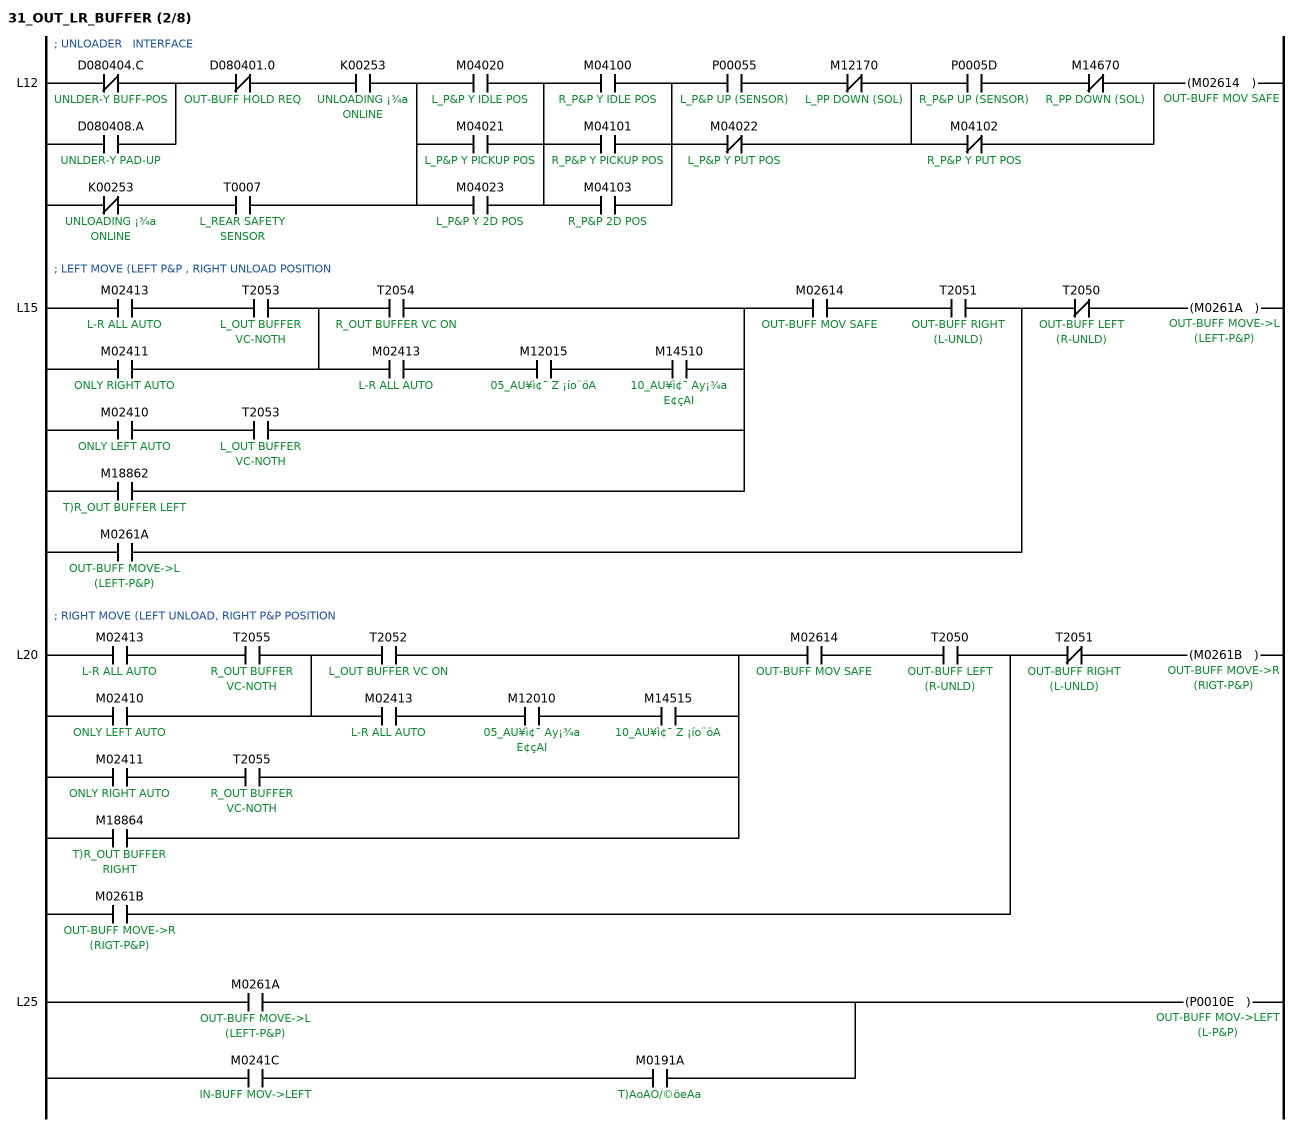
[picture p216: 31_OUT_LR_BUFFER rungs L12-L25]
//  UNLOADER   INTERFACE
; L12
LOAD NOT  D080404.C	// UNLDER-Y BUFF-POS
OR        D080408.A	// UNLDER-Y PAD-UP
AND NOT   D080401.0	// OUT-BUFF HOLD REQ
AND       K00253	// UNLOADING ¡¾a ONLINE
LOAD NOT  K00253	// UNLOADING ¡¾a ONLINE
AND       T0007	// L_REAR SAFETY SENSOR
OR LOAD
LOAD      M04020	// L_P&P Y IDLE POS
OR        M04021	// L_P&P Y PICKUP POS
OR        M04023	// L_P&P Y 2D POS
AND LOAD
LOAD      M04100	// R_P&P Y IDLE POS
OR        M04101	// R_P&P Y PICKUP POS
OR        M04103	// R_P&P 2D POS
AND LOAD
LOAD      P00055	// L_P&P UP (SENSOR)
AND NOT   M12170	// L_PP DOWN (SOL)
OR NOT    M04022	// L_P&P Y PUT POS
AND LOAD
LOAD      P0005D	// R_P&P UP (SENSOR)
AND NOT   M14670	// R_PP DOWN (SOL)
OR NOT    M04102	// R_P&P Y PUT POS
AND LOAD
OUT       M02614	// OUT-BUFF MOV SAFE
; L15
LOAD      M02413	// L-R ALL AUTO
AND       T2053	// L_OUT BUFFER VC-NOTH
OR        M02411	// ONLY RIGHT AUTO
LOAD      T2054	// R_OUT BUFFER VC ON
LOAD      M02413	// L-R ALL AUTO
AND       M12015	// 05_AU¥ì¢¯ Z ¡ío¨öA
AND       M14510	// 10_AU¥ì¢¯ Ay¡¾a E¢çAI
OR LOAD
AND LOAD
LOAD      M02410	// ONLY LEFT AUTO
AND       T2053	// L_OUT BUFFER VC-NOTH
OR LOAD
OR        M18862	// T)R_OUT BUFFER LEFT
AND       M02614	// OUT-BUFF MOV SAFE
AND       T2051	// OUT-BUFF RIGHT (L-UNLD)
OR        M0261A	// OUT-BUFF MOVE->L (LEFT-P&P)
AND NOT   T2050	// OUT-BUFF LEFT (R-UNLD)
OUT       M0261A	// OUT-BUFF MOVE->L (LEFT-P&P)
// output comment: LEFT MOVE (LEFT P&P , RIGHT UNLOAD POSITION
; L20
LOAD      M02413	// L-R ALL AUTO
AND       T2055	// R_OUT BUFFER VC-NOTH
OR        M02410	// ONLY LEFT AUTO
LOAD      T2052	// L_OUT BUFFER VC ON
LOAD      M02413	// L-R ALL AUTO
AND       M12010	// 05_AU¥ì¢¯ Ay¡¾a E¢çAI
AND       M14515	// 10_AU¥ì¢¯ Z ¡ío¨öA
OR LOAD
AND LOAD
LOAD      M02411	// ONLY RIGHT AUTO
AND       T2055	// R_OUT BUFFER VC-NOTH
OR LOAD
OR        M18864	// T)R_OUT BUFFER RIGHT
AND       M02614	// OUT-BUFF MOV SAFE
AND       T2050	// OUT-BUFF LEFT (R-UNLD)
OR        M0261B	// OUT-BUFF MOVE->R (RIGT-P&P)
AND NOT   T2051	// OUT-BUFF RIGHT (L-UNLD)
OUT       M0261B	// OUT-BUFF MOVE->R (RIGT-P&P)
// output comment: RIGHT MOVE (LEFT UNLOAD, RIGHT P&P POSITION
; L25
LOAD      M0261A	// OUT-BUFF MOVE->L (LEFT-P&P)
LOAD      M0241C	// IN-BUFF MOV->LEFT
AND       M0191A	// T)AoAO/©öeAa
OR LOAD
OUT       P0010E	// OUT-BUFF MOV->LEFT (L-P&P)

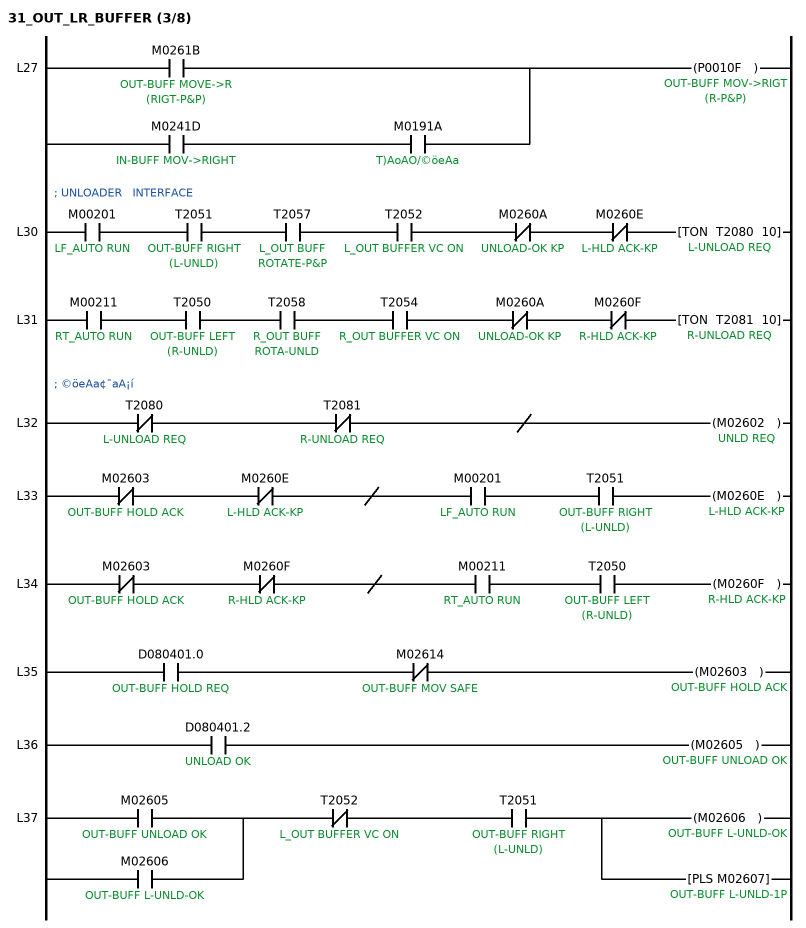
; L27
LOAD      M0261B	// OUT-BUFF MOVE->R (RIGT-P&P)
LOAD      M0241D	// IN-BUFF MOV->RIGHT
AND       M0191A	// T)AoAO/©öeAa
OR LOAD
OUT       P0010F	// OUT-BUFF MOV->RIGT (R-P&P)
//  UNLOADER   INTERFACE
; L30
LOAD      M00201	// LF_AUTO RUN
AND       T2051	// OUT-BUFF RIGHT (L-UNLD)
AND       T2057	// L_OUT BUFF ROTATE-P&P
AND       T2052	// L_OUT BUFFER VC ON
AND NOT   M0260A	// UNLOAD-OK KP
AND NOT   M0260E	// L-HLD ACK-KP
TON       T2080 10	// L-UNLOAD REQ
; L31
LOAD      M00211	// RT_AUTO RUN
AND       T2050	// OUT-BUFF LEFT (R-UNLD)
AND       T2058	// R_OUT BUFF ROTA-UNLD
AND       T2054	// R_OUT BUFFER VC ON
AND NOT   M0260A	// UNLOAD-OK KP
AND NOT   M0260F	// R-HLD ACK-KP
TON       T2081 10	// R-UNLOAD REQ
; L32
LOAD NOT  T2080	// L-UNLOAD REQ
AND NOT   T2081	// R-UNLOAD REQ
NOT
OUT       M02602	// UNLD REQ
// output comment: ©öeAa¢¯aA¡í
; L33
LOAD NOT  M02603	// OUT-BUFF HOLD ACK
AND NOT   M0260E	// L-HLD ACK-KP
NOT
AND       M00201	// LF_AUTO RUN
AND       T2051	// OUT-BUFF RIGHT (L-UNLD)
OUT       M0260E	// L-HLD ACK-KP
; L34
LOAD NOT  M02603	// OUT-BUFF HOLD ACK
AND NOT   M0260F	// R-HLD ACK-KP
NOT
AND       M00211	// RT_AUTO RUN
AND       T2050	// OUT-BUFF LEFT (R-UNLD)
OUT       M0260F	// R-HLD ACK-KP
; L35
LOAD      D080401.0	// OUT-BUFF HOLD REQ
AND NOT   M02614	// OUT-BUFF MOV SAFE
OUT       M02603	// OUT-BUFF HOLD ACK
; L36
LOAD      D080401.2	// UNLOAD OK
OUT       M02605	// OUT-BUFF UNLOAD OK
; L37
LOAD      M02605	// OUT-BUFF UNLOAD OK
OR        M02606	// OUT-BUFF L-UNLD-OK
AND NOT   T2052	// L_OUT BUFFER VC ON
AND       T2051	// OUT-BUFF RIGHT (L-UNLD)
OUT       M02606	// OUT-BUFF L-UNLD-OK
OUTP      M02607	// OUT-BUFF L-UNLD-1P

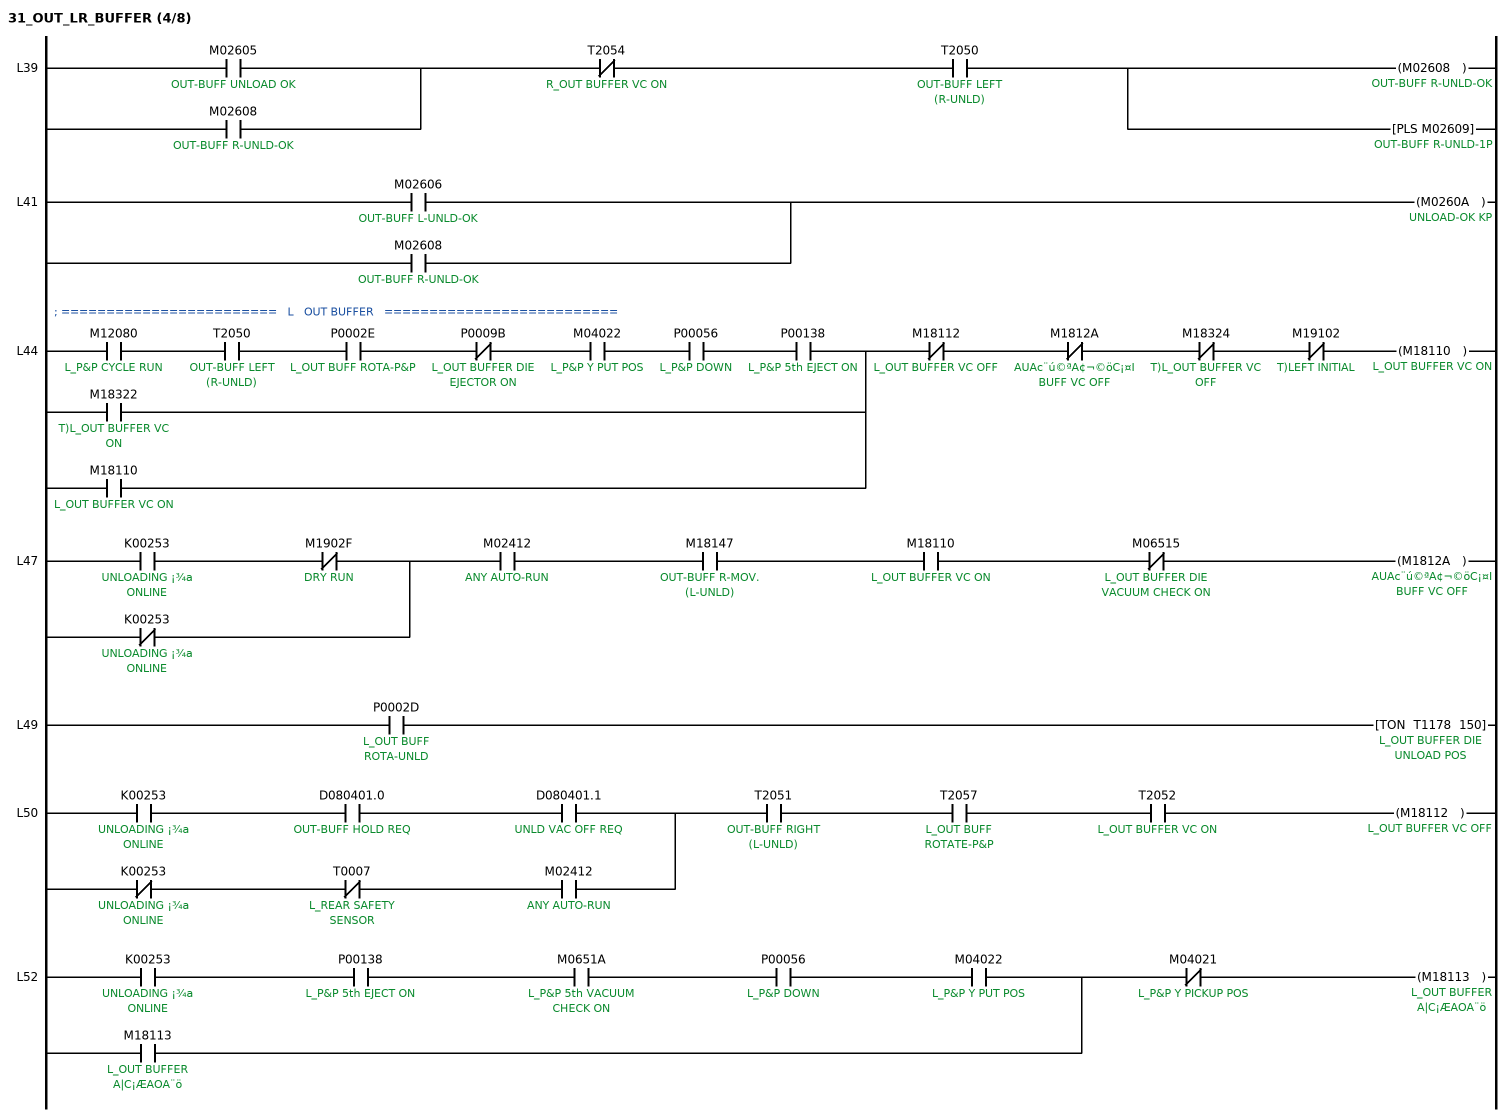
; L39
LOAD      M02605	// OUT-BUFF UNLOAD OK
OR        M02608	// OUT-BUFF R-UNLD-OK
AND NOT   T2054	// R_OUT BUFFER VC ON
AND       T2050	// OUT-BUFF LEFT (R-UNLD)
OUT       M02608	// OUT-BUFF R-UNLD-OK
OUTP      M02609	// OUT-BUFF R-UNLD-1P
; L41
LOAD      M02606	// OUT-BUFF L-UNLD-OK
OR        M02608	// OUT-BUFF R-UNLD-OK
OUT       M0260A	// UNLOAD-OK KP
// ========================   L   OUT BUFFER   ==========================
; L44
LOAD      M12080	// L_P&P CYCLE RUN
AND       T2050	// OUT-BUFF LEFT (R-UNLD)
AND       P0002E	// L_OUT BUFF ROTA-P&P
AND NOT   P0009B	// L_OUT BUFFER DIE EJECTOR ON
AND       M04022	// L_P&P Y PUT POS
AND       P00056	// L_P&P DOWN
AND       P00138	// L_P&P 5th EJECT ON
OR        M18322	// T)L_OUT BUFFER VC ON
OR        M18110	// L_OUT BUFFER VC ON
AND NOT   M18112	// L_OUT BUFFER VC OFF
AND NOT   M1812A	// AUAc¨ú©ªA¢¬©öC¡¤I BUFF VC OFF
AND NOT   M18324	// T)L_OUT BUFFER VC OFF
AND NOT   M19102	// T)LEFT INITIAL
OUT       M18110	// L_OUT BUFFER VC ON
; L47
LOAD      K00253	// UNLOADING ¡¾a ONLINE
AND NOT   M1902F	// DRY RUN
OR NOT    K00253	// UNLOADING ¡¾a ONLINE
AND       M02412	// ANY AUTO-RUN
AND       M18147	// OUT-BUFF R-MOV.  (L-UNLD)
AND       M18110	// L_OUT BUFFER VC ON
AND NOT   M06515	// L_OUT BUFFER DIE VACUUM CHECK ON
OUT       M1812A	// AUAc¨ú©ªA¢¬©öC¡¤I BUFF VC OFF
; L49
LOAD      P0002D	// L_OUT BUFF ROTA-UNLD
TON       T1178 150	// L_OUT BUFFER DIE UNLOAD POS
; L50
LOAD      K00253	// UNLOADING ¡¾a ONLINE
AND       D080401.0	// OUT-BUFF HOLD REQ
AND       D080401.1	// UNLD VAC OFF REQ
LOAD NOT  K00253	// UNLOADING ¡¾a ONLINE
AND NOT   T0007	// L_REAR SAFETY SENSOR
AND       M02412	// ANY AUTO-RUN
OR LOAD
AND       T2051	// OUT-BUFF RIGHT (L-UNLD)
AND       T2057	// L_OUT BUFF ROTATE-P&P
AND       T2052	// L_OUT BUFFER VC ON
OUT       M18112	// L_OUT BUFFER VC OFF
; L52
LOAD      K00253	// UNLOADING ¡¾a ONLINE
AND       P00138	// L_P&P 5th EJECT ON
AND       M0651A	// L_P&P 5th VACUUM CHECK ON
AND       P00056	// L_P&P DOWN
AND       M04022	// L_P&P Y PUT POS
OR        M18113	// L_OUT BUFFER A|C¡ÆAOA¨ö
AND NOT   M04021	// L_P&P Y PICKUP POS
OUT       M18113	// L_OUT BUFFER A|C¡ÆAOA¨ö

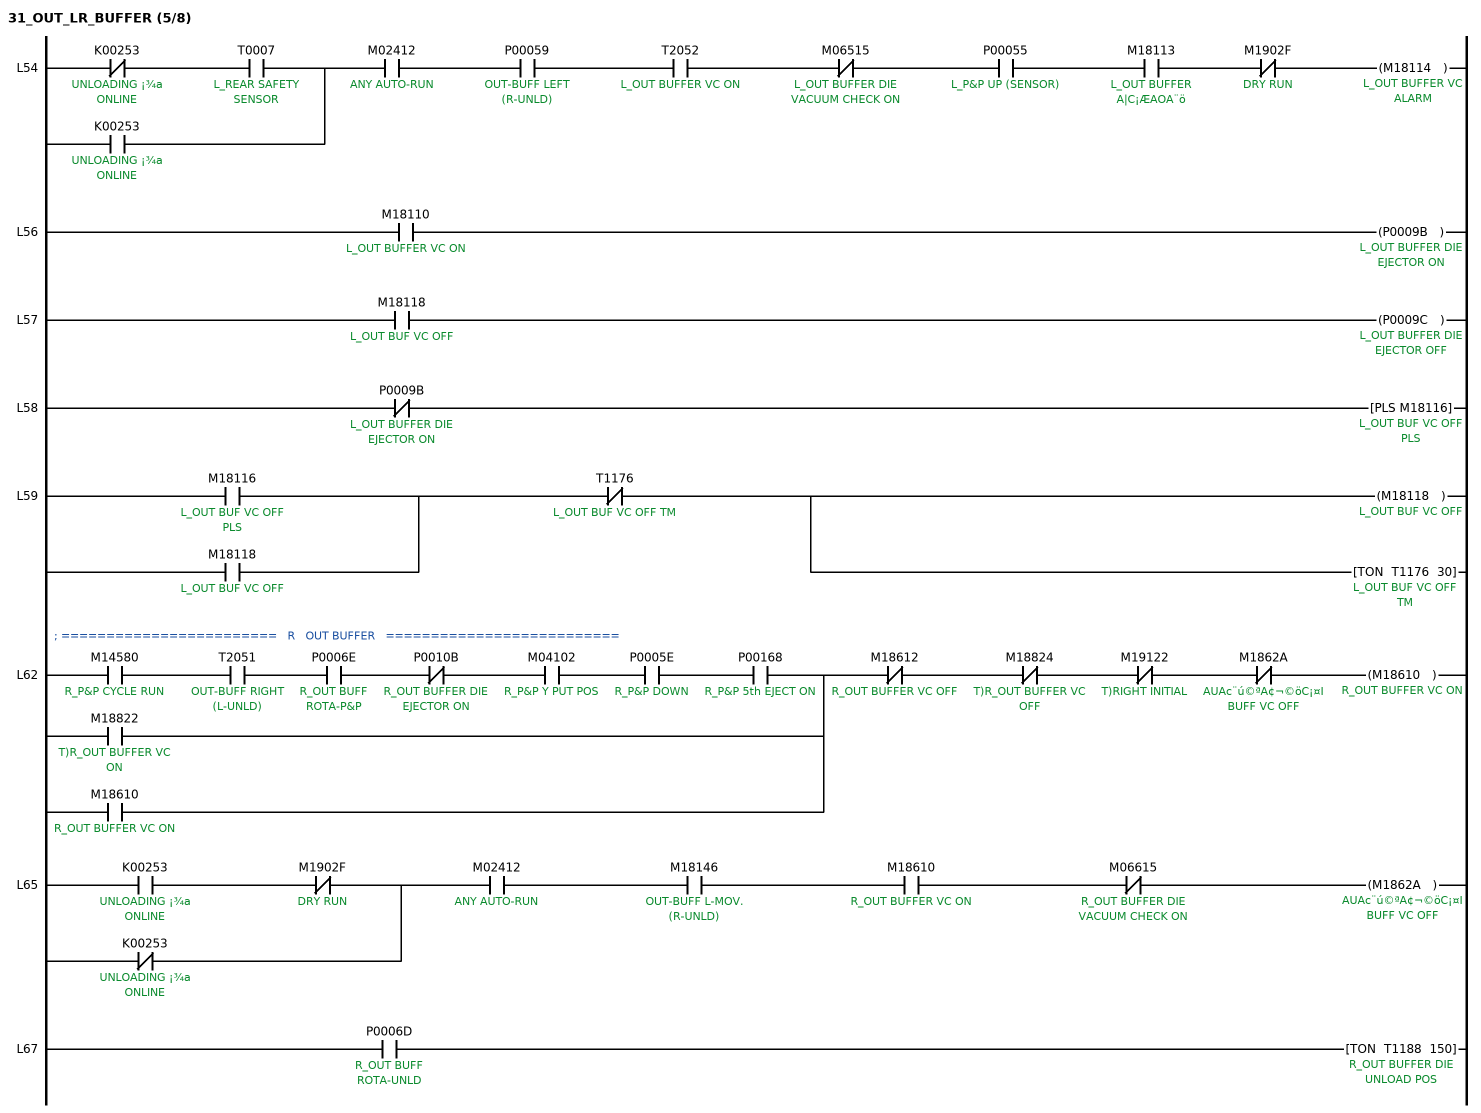
; L54
LOAD NOT  K00253	// UNLOADING ¡¾a ONLINE
AND       T0007	// L_REAR SAFETY SENSOR
OR        K00253	// UNLOADING ¡¾a ONLINE
AND       M02412	// ANY AUTO-RUN
AND       P00059	// OUT-BUFF LEFT (R-UNLD)
AND       T2052	// L_OUT BUFFER VC ON
AND NOT   M06515	// L_OUT BUFFER DIE VACUUM CHECK ON
AND       P00055	// L_P&P UP (SENSOR)
AND       M18113	// L_OUT BUFFER A|C¡ÆAOA¨ö
AND NOT   M1902F	// DRY RUN
OUT       M18114	// L_OUT BUFFER VC ALARM
; L56
LOAD      M18110	// L_OUT BUFFER VC ON
OUT       P0009B	// L_OUT BUFFER DIE EJECTOR ON
; L57
LOAD      M18118	// L_OUT BUF VC OFF
OUT       P0009C	// L_OUT BUFFER DIE EJECTOR OFF
; L58
LOAD NOT  P0009B	// L_OUT BUFFER DIE EJECTOR ON
OUTP      M18116	// L_OUT BUF VC OFF PLS
; L59
LOAD      M18116	// L_OUT BUF VC OFF PLS
OR        M18118	// L_OUT BUF VC OFF
AND NOT   T1176	// L_OUT BUF VC OFF TM
OUT       M18118	// L_OUT BUF VC OFF
TON       T1176 30	// L_OUT BUF VC OFF TM
// ========================   R   OUT BUFFER   ==========================
; L62
LOAD      M14580	// R_P&P CYCLE RUN
AND       T2051	// OUT-BUFF RIGHT (L-UNLD)
AND       P0006E	// R_OUT BUFF ROTA-P&P
AND NOT   P0010B	// R_OUT BUFFER DIE EJECTOR ON
AND       M04102	// R_P&P Y PUT POS
AND       P0005E	// R_P&P DOWN
AND       P00168	// R_P&P 5th EJECT ON
OR        M18822	// T)R_OUT BUFFER VC ON
OR        M18610	// R_OUT BUFFER VC ON
AND NOT   M18612	// R_OUT BUFFER VC OFF
AND NOT   M18824	// T)R_OUT BUFFER VC OFF
AND NOT   M19122	// T)RIGHT INITIAL
AND NOT   M1862A	// AUAc¨ú©ªA¢¬©öC¡¤I BUFF VC OFF
OUT       M18610	// R_OUT BUFFER VC ON
; L65
LOAD      K00253	// UNLOADING ¡¾a ONLINE
AND NOT   M1902F	// DRY RUN
OR NOT    K00253	// UNLOADING ¡¾a ONLINE
AND       M02412	// ANY AUTO-RUN
AND       M18146	// OUT-BUFF L-MOV.  (R-UNLD)
AND       M18610	// R_OUT BUFFER VC ON
AND NOT   M06615	// R_OUT BUFFER DIE VACUUM CHECK ON
OUT       M1862A	// AUAc¨ú©ªA¢¬©öC¡¤I BUFF VC OFF
; L67
LOAD      P0006D	// R_OUT BUFF ROTA-UNLD
TON       T1188 150	// R_OUT BUFFER DIE UNLOAD POS

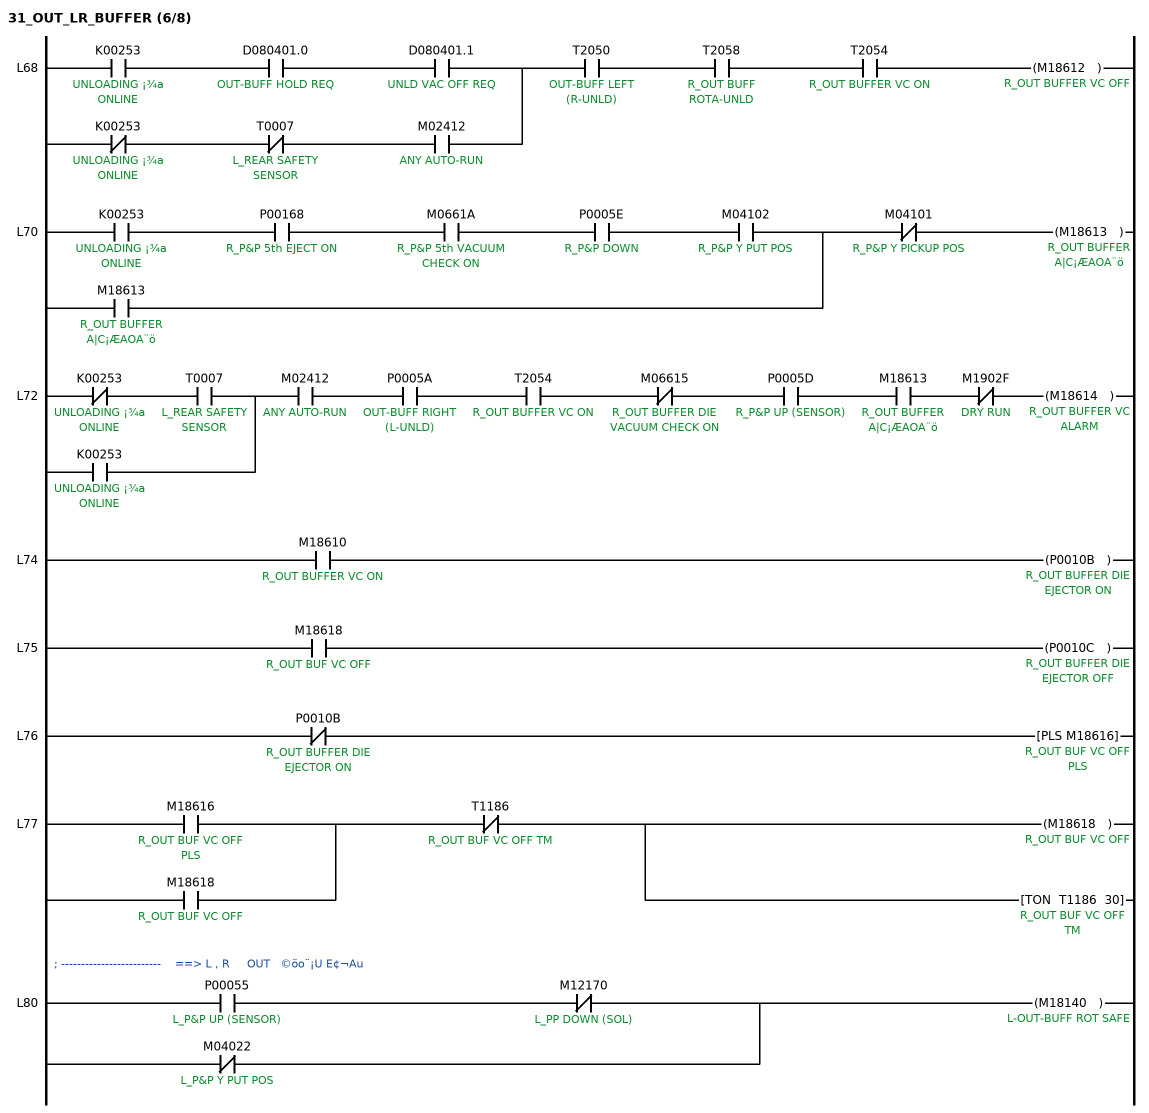
; L68
LOAD      K00253	// UNLOADING ¡¾a ONLINE
AND       D080401.0	// OUT-BUFF HOLD REQ
AND       D080401.1	// UNLD VAC OFF REQ
LOAD NOT  K00253	// UNLOADING ¡¾a ONLINE
AND NOT   T0007	// L_REAR SAFETY SENSOR
AND       M02412	// ANY AUTO-RUN
OR LOAD
AND       T2050	// OUT-BUFF LEFT (R-UNLD)
AND       T2058	// R_OUT BUFF ROTA-UNLD
AND       T2054	// R_OUT BUFFER VC ON
OUT       M18612	// R_OUT BUFFER VC OFF
; L70
LOAD      K00253	// UNLOADING ¡¾a ONLINE
AND       P00168	// R_P&P 5th EJECT ON
AND       M0661A	// R_P&P 5th VACUUM CHECK ON
AND       P0005E	// R_P&P DOWN
AND       M04102	// R_P&P Y PUT POS
OR        M18613	// R_OUT BUFFER A|C¡ÆAOA¨ö
AND NOT   M04101	// R_P&P Y PICKUP POS
OUT       M18613	// R_OUT BUFFER A|C¡ÆAOA¨ö
; L72
LOAD NOT  K00253	// UNLOADING ¡¾a ONLINE
AND       T0007	// L_REAR SAFETY SENSOR
OR        K00253	// UNLOADING ¡¾a ONLINE
AND       M02412	// ANY AUTO-RUN
AND       P0005A	// OUT-BUFF RIGHT (L-UNLD)
AND       T2054	// R_OUT BUFFER VC ON
AND NOT   M06615	// R_OUT BUFFER DIE VACUUM CHECK ON
AND       P0005D	// R_P&P UP (SENSOR)
AND       M18613	// R_OUT BUFFER A|C¡ÆAOA¨ö
AND NOT   M1902F	// DRY RUN
OUT       M18614	// R_OUT BUFFER VC ALARM
; L74
LOAD      M18610	// R_OUT BUFFER VC ON
OUT       P0010B	// R_OUT BUFFER DIE EJECTOR ON
; L75
LOAD      M18618	// R_OUT BUF VC OFF
OUT       P0010C	// R_OUT BUFFER DIE EJECTOR OFF
; L76
LOAD NOT  P0010B	// R_OUT BUFFER DIE EJECTOR ON
OUTP      M18616	// R_OUT BUF VC OFF PLS
; L77
LOAD      M18616	// R_OUT BUF VC OFF PLS
OR        M18618	// R_OUT BUF VC OFF
AND NOT   T1186	// R_OUT BUF VC OFF TM
OUT       M18618	// R_OUT BUF VC OFF
TON       T1186 30	// R_OUT BUF VC OFF TM
// -------------------------    ==> L , R     OUT   ©öo¨¡U E¢¬Au
; L80
LOAD      P00055	// L_P&P UP (SENSOR)
AND NOT   M12170	// L_PP DOWN (SOL)
OR NOT    M04022	// L_P&P Y PUT POS
OUT       M18140	// L-OUT-BUFF ROT SAFE

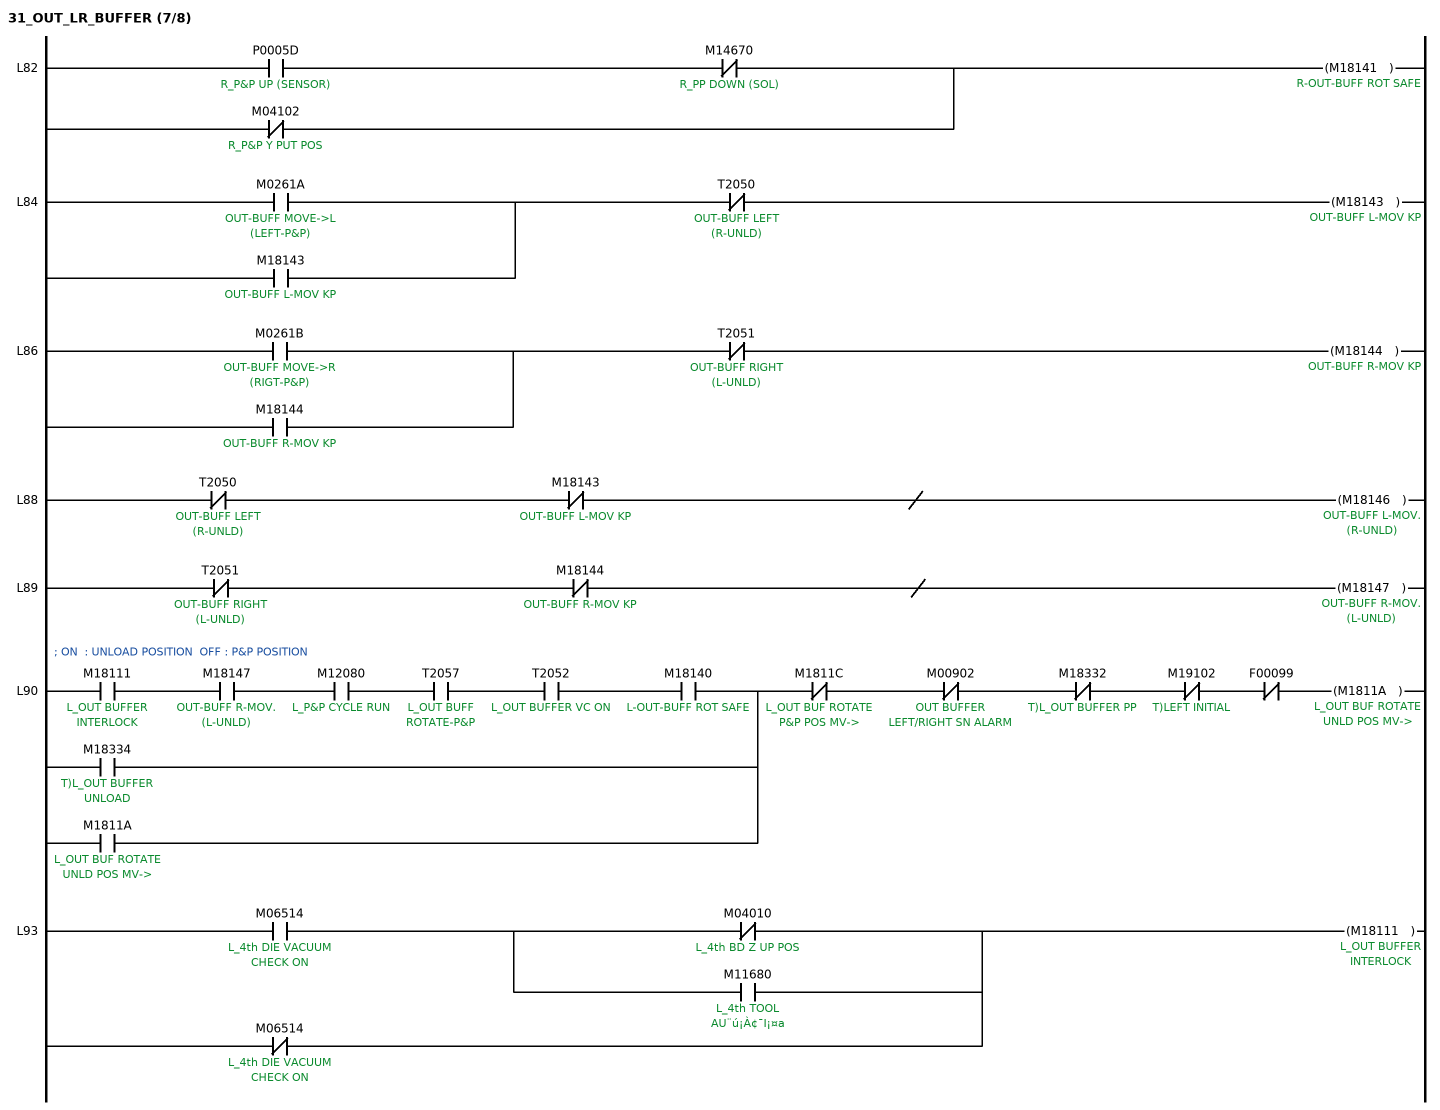
; L82
LOAD      P0005D	// R_P&P UP (SENSOR)
AND NOT   M14670	// R_PP DOWN (SOL)
OR NOT    M04102	// R_P&P Y PUT POS
OUT       M18141	// R-OUT-BUFF ROT SAFE
; L84
LOAD      M0261A	// OUT-BUFF MOVE->L (LEFT-P&P)
OR        M18143	// OUT-BUFF L-MOV KP
AND NOT   T2050	// OUT-BUFF LEFT (R-UNLD)
OUT       M18143	// OUT-BUFF L-MOV KP
; L86
LOAD      M0261B	// OUT-BUFF MOVE->R (RIGT-P&P)
OR        M18144	// OUT-BUFF R-MOV KP
AND NOT   T2051	// OUT-BUFF RIGHT (L-UNLD)
OUT       M18144	// OUT-BUFF R-MOV KP
; L88
LOAD NOT  T2050	// OUT-BUFF LEFT (R-UNLD)
AND NOT   M18143	// OUT-BUFF L-MOV KP
NOT
OUT       M18146	// OUT-BUFF L-MOV.  (R-UNLD)
; L89
LOAD NOT  T2051	// OUT-BUFF RIGHT (L-UNLD)
AND NOT   M18144	// OUT-BUFF R-MOV KP
NOT
OUT       M18147	// OUT-BUFF R-MOV.  (L-UNLD)
; L90
LOAD      M18111	// L_OUT BUFFER INTERLOCK
AND       M18147	// OUT-BUFF R-MOV.  (L-UNLD)
AND       M12080	// L_P&P CYCLE RUN
AND       T2057	// L_OUT BUFF ROTATE-P&P
AND       T2052	// L_OUT BUFFER VC ON
AND       M18140	// L-OUT-BUFF ROT SAFE
OR        M18334	// T)L_OUT BUFFER UNLOAD
OR        M1811A	// L_OUT BUF ROTATE UNLD POS MV->
AND NOT   M1811C	// L_OUT BUF ROTATE P&P POS MV->
AND NOT   M00902	// OUT BUFFER LEFT/RIGHT SN ALARM
AND NOT   M18332	// T)L_OUT BUFFER PP
AND NOT   M19102	// T)LEFT INITIAL
AND NOT   F00099
OUT       M1811A	// L_OUT BUF ROTATE UNLD POS MV->
// output comment: ON  : UNLOAD POSITION  OFF : P&P POSITION
; L93
LOAD      M06514	// L_4th DIE VACUUM CHECK ON
LOAD NOT  M04010	// L_4th BD Z UP POS
OR        M11680	// L_4th TOOL AU¨ú¡À¢¯I¡¤a
AND LOAD
OR NOT    M06514	// L_4th DIE VACUUM CHECK ON
OUT       M18111	// L_OUT BUFFER INTERLOCK

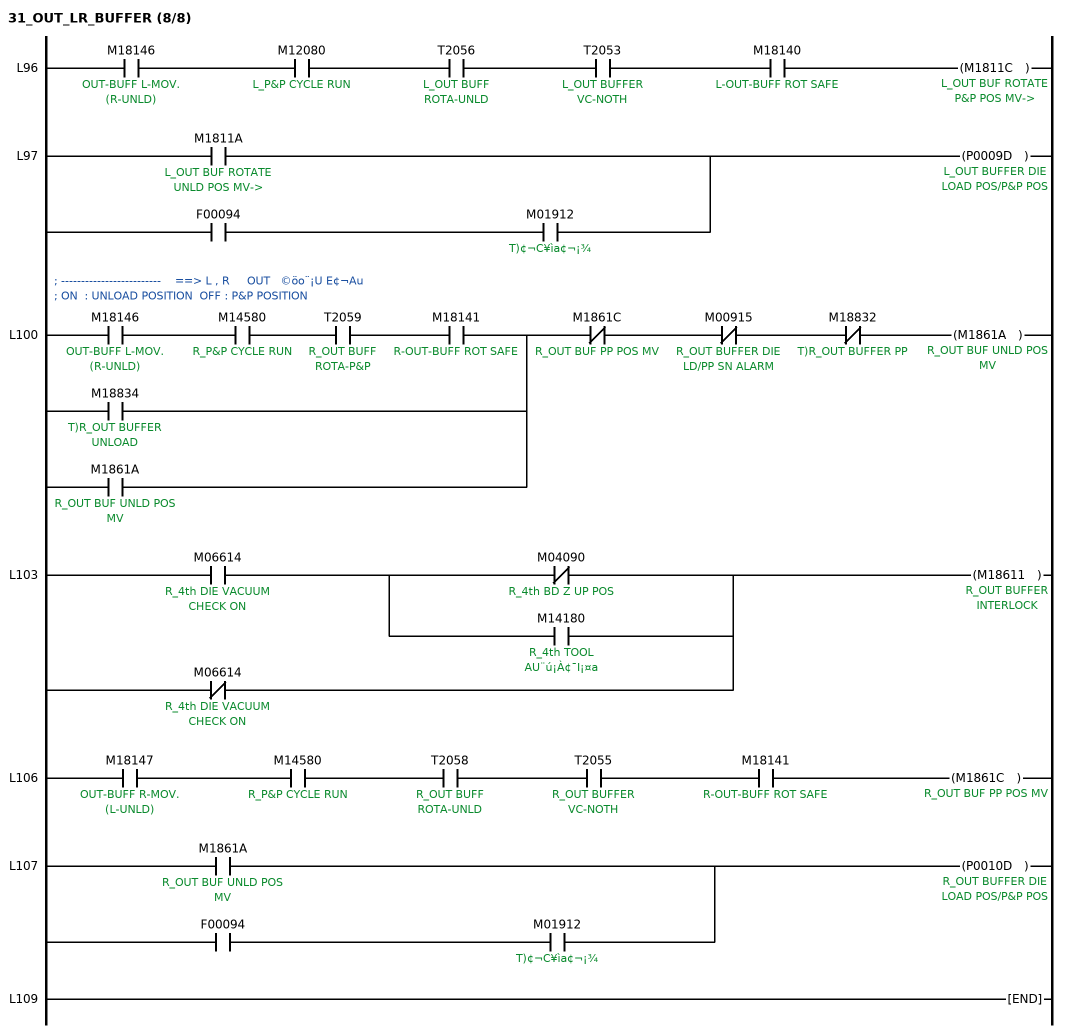
; L96
LOAD      M18146	// OUT-BUFF L-MOV.  (R-UNLD)
AND       M12080	// L_P&P CYCLE RUN
AND       T2056	// L_OUT BUFF ROTA-UNLD
AND       T2053	// L_OUT BUFFER VC-NOTH
AND       M18140	// L-OUT-BUFF ROT SAFE
OUT       M1811C	// L_OUT BUF ROTATE P&P POS MV->
; L97
LOAD      M1811A	// L_OUT BUF ROTATE UNLD POS MV->
LOAD      F00094
AND       M01912	// T)¢¬C¥ìa¢¬¡¾
OR LOAD
OUT       P0009D	// L_OUT BUFFER DIE LOAD POS/P&P POS
// -------------------------    ==> L , R     OUT   ©öo¨¡U E¢¬Au
; L100
LOAD      M18146	// OUT-BUFF L-MOV.  (R-UNLD)
AND       M14580	// R_P&P CYCLE RUN
AND       T2059	// R_OUT BUFF ROTA-P&P
AND       M18141	// R-OUT-BUFF ROT SAFE
OR        M18834	// T)R_OUT BUFFER UNLOAD
OR        M1861A	// R_OUT BUF UNLD POS MV
AND NOT   M1861C	// R_OUT BUF PP POS MV
AND NOT   M00915	// R_OUT BUFFER DIE LD/PP SN ALARM
AND NOT   M18832	// T)R_OUT BUFFER PP
OUT       M1861A	// R_OUT BUF UNLD POS MV
// output comment: ON  : UNLOAD POSITION  OFF : P&P POSITION
; L103
LOAD      M06614	// R_4th DIE VACUUM CHECK ON
LOAD NOT  M04090	// R_4th BD Z UP POS
OR        M14180	// R_4th TOOL AU¨ú¡À¢¯I¡¤a
AND LOAD
OR NOT    M06614	// R_4th DIE VACUUM CHECK ON
OUT       M18611	// R_OUT BUFFER INTERLOCK
; L106
LOAD      M18147	// OUT-BUFF R-MOV.  (L-UNLD)
AND       M14580	// R_P&P CYCLE RUN
AND       T2058	// R_OUT BUFF ROTA-UNLD
AND       T2055	// R_OUT BUFFER VC-NOTH
AND       M18141	// R-OUT-BUFF ROT SAFE
OUT       M1861C	// R_OUT BUF PP POS MV
; L107
LOAD      M1861A	// R_OUT BUF UNLD POS MV
LOAD      F00094
AND       M01912	// T)¢¬C¥ìa¢¬¡¾
OR LOAD
OUT       P0010D	// R_OUT BUFFER DIE LOAD POS/P&P POS
; L109
END

PROGRAM 40_2D_CODE (task: ¨ö¨¬A¥ì CA¡¤I¡¾¡¿¡¤¡Í)

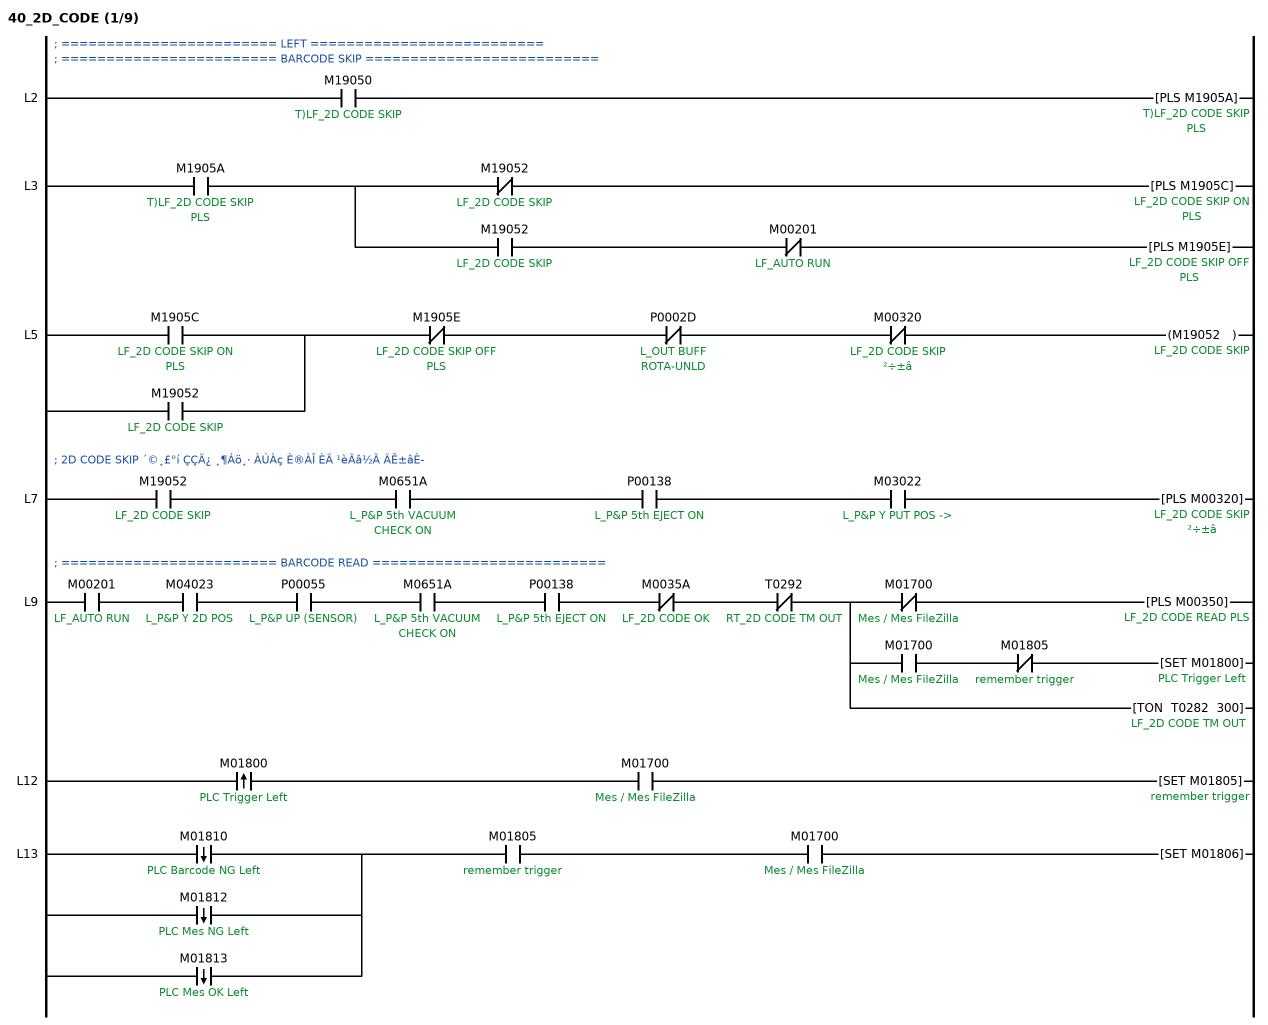
// ======================== LEFT ==========================
// ======================== BARCODE SKIP ==========================
; L2
LOAD      M19050	// T)LF_2D CODE SKIP
OUTP      M1905A	// T)LF_2D CODE SKIP PLS
; L3
LOAD      M1905A	// T)LF_2D CODE SKIP PLS
MPUSH
AND NOT   M19052	// LF_2D CODE SKIP
OUTP      M1905C	// LF_2D CODE SKIP ON PLS
MPOP
AND       M19052	// LF_2D CODE SKIP
AND NOT   M00201	// LF_AUTO RUN
OUTP      M1905E	// LF_2D CODE SKIP OFF PLS
; L5
LOAD      M1905C	// LF_2D CODE SKIP ON PLS
OR        M19052	// LF_2D CODE SKIP
AND NOT   M1905E	// LF_2D CODE SKIP OFF PLS
AND NOT   P0002D	// L_OUT BUFF ROTA-UNLD
AND NOT   M00320	// LF_2D CODE SKIP ²÷±â
OUT       M19052	// LF_2D CODE SKIP
; L7
LOAD      M19052	// LF_2D CODE SKIP
AND       M0651A	// L_P&P 5th VACUUM CHECK ON
AND       P00138	// L_P&P 5th EJECT ON
AND       M03022	// L_P&P Y PUT POS ->
OUTP      M00320	// LF_2D CODE SKIP ²÷±â
// output comment: 2D CODE SKIP ´©¸£°í ÇÇÄ¿ ¸¶Áö¸· ÀÚÀç È®ÀÎ ÈÄ ¹èÃâ½Ã ÃÊ±âÈ­
// ======================== BARCODE READ ==========================
; L9
LOAD      M00201	// LF_AUTO RUN
AND       M04023	// L_P&P Y 2D POS
AND       P00055	// L_P&P UP (SENSOR)
AND       M0651A	// L_P&P 5th VACUUM CHECK ON
AND       P00138	// L_P&P 5th EJECT ON
AND NOT   M0035A	// LF_2D CODE OK
AND NOT   T0292	// RT_2D CODE TM OUT
MPUSH
AND NOT   M01700	// Mes / Mes FileZilla
OUTP      M00350	// LF_2D CODE READ PLS
MLOAD
AND       M01700	// Mes / Mes FileZilla
AND NOT   M01805	// remember trigger
SET       M01800	// PLC Trigger Left
MPOP
TON       T0282 300	// LF_2D CODE TM OUT
; L12
LOADP     M01800	// PLC Trigger Left
AND       M01700	// Mes / Mes FileZilla
SET       M01805	// remember trigger
; L13
LOADN     M01810	// PLC Barcode NG Left
ORN       M01812	// PLC Mes NG Left
ORN       M01813	// PLC Mes OK Left
AND       M01805	// remember trigger
AND       M01700	// Mes / Mes FileZilla
SET       M01806

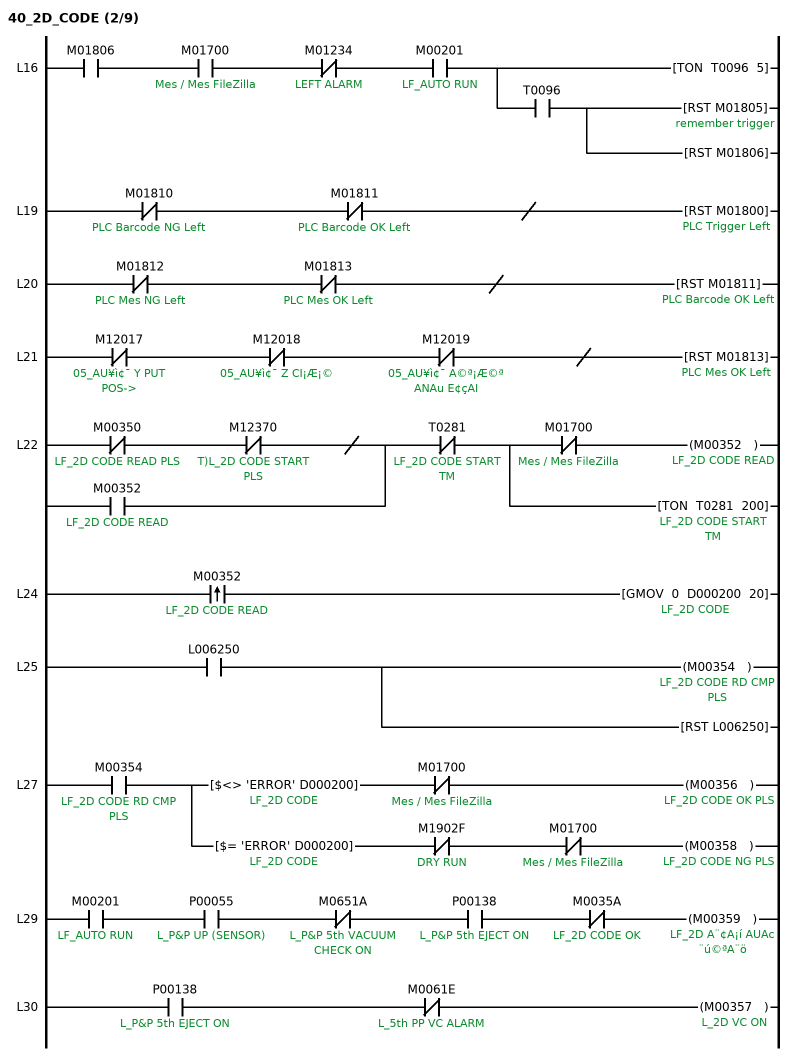
; L16
LOAD      M01806
AND       M01700	// Mes / Mes FileZilla
AND NOT   M01234	// LEFT ALARM
AND       M00201	// LF_AUTO RUN
TON       T0096 5
AND       T0096
RST       M01805	// remember trigger
RST       M01806
; L19
LOAD NOT  M01810	// PLC Barcode NG Left
AND NOT   M01811	// PLC Barcode OK Left
NOT
RST       M01800	// PLC Trigger Left
; L20
LOAD NOT  M01812	// PLC Mes NG Left
AND NOT   M01813	// PLC Mes OK Left
NOT
RST       M01811	// PLC Barcode OK Left
; L21
LOAD NOT  M12017	// 05_AU¥ì¢¯ Y PUT POS->
AND NOT   M12018	// 05_AU¥ì¢¯ Z CI¡Æ¡©
AND NOT   M12019	// 05_AU¥ì¢¯ A©ª¡Æ©ª ANAu E¢çAI
NOT
RST       M01813	// PLC Mes OK Left
; L22
LOAD NOT  M00350	// LF_2D CODE READ PLS
AND NOT   M12370	// T)L_2D CODE START PLS
NOT
OR        M00352	// LF_2D CODE READ
AND NOT   T0281	// LF_2D CODE START TM
MPUSH
AND NOT   M01700	// Mes / Mes FileZilla
OUT       M00352	// LF_2D CODE READ
MPOP
TON       T0281 200	// LF_2D CODE START TM
; L24
LOADP     M00352	// LF_2D CODE READ
GMOV      0 D000200 20	// LF_2D CODE
; L25
LOAD      L006250
OUT       M00354	// LF_2D CODE RD CMP PLS
RST       L006250
; L27
LOAD      M00354	// LF_2D CODE RD CMP PLS
MPUSH
AND$<>    'ERROR' D000200	// LF_2D CODE
AND NOT   M01700	// Mes / Mes FileZilla
OUT       M00356	// LF_2D CODE OK PLS
MPOP
AND$=     'ERROR' D000200	// LF_2D CODE
AND NOT   M1902F	// DRY RUN
AND NOT   M01700	// Mes / Mes FileZilla
OUT       M00358	// LF_2D CODE NG PLS
; L29
LOAD      M00201	// LF_AUTO RUN
AND       P00055	// L_P&P UP (SENSOR)
AND NOT   M0651A	// L_P&P 5th VACUUM CHECK ON
AND       P00138	// L_P&P 5th EJECT ON
AND NOT   M0035A	// LF_2D CODE OK
OUT       M00359	// LF_2D A¨¢A¡í AUAc ¨ú©ªA¨ö
; L30
LOAD      P00138	// L_P&P 5th EJECT ON
AND NOT   M0061E	// L_5th PP VC ALARM
OUT       M00357	// L_2D VC ON

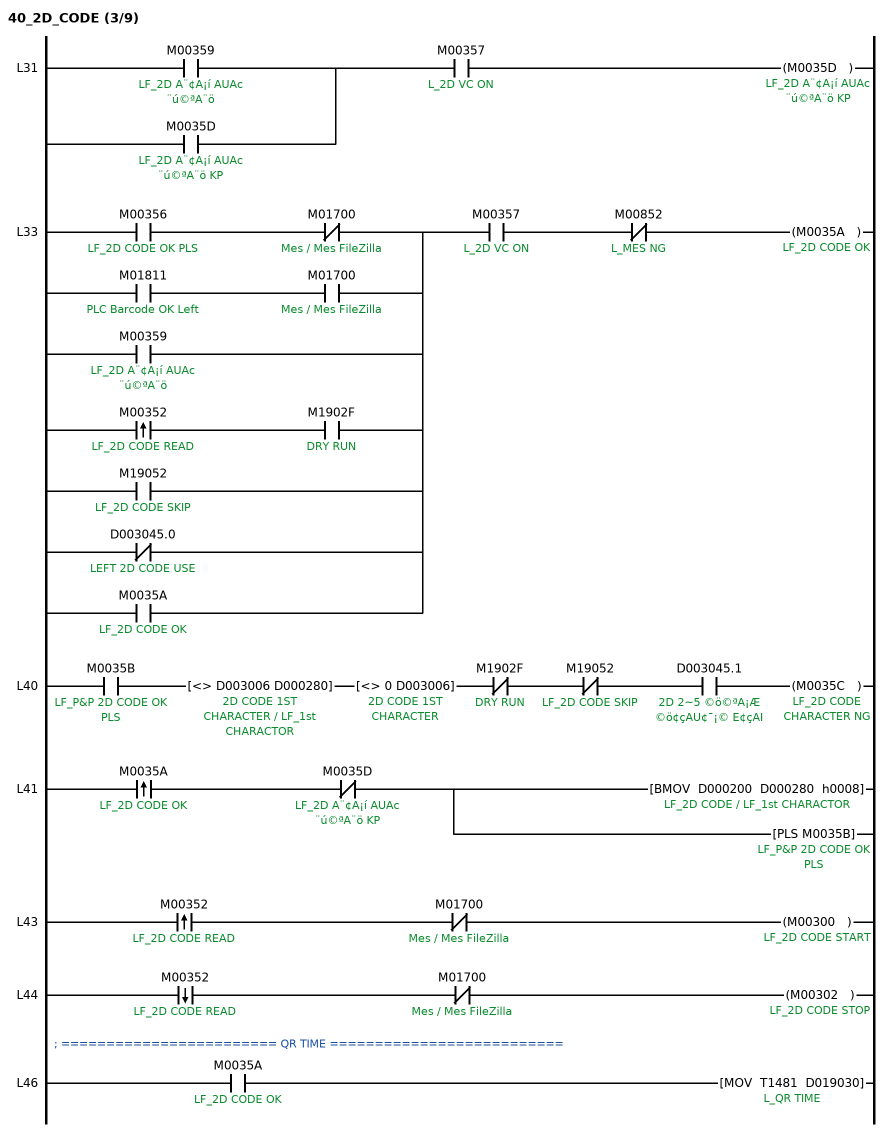
; L31
LOAD      M00359	// LF_2D A¨¢A¡í AUAc ¨ú©ªA¨ö
OR        M0035D	// LF_2D A¨¢A¡í AUAc ¨ú©ªA¨ö KP
AND       M00357	// L_2D VC ON
OUT       M0035D	// LF_2D A¨¢A¡í AUAc ¨ú©ªA¨ö KP
; L33
LOAD      M00356	// LF_2D CODE OK PLS
AND NOT   M01700	// Mes / Mes FileZilla
LOAD      M01811	// PLC Barcode OK Left
AND       M01700	// Mes / Mes FileZilla
OR LOAD
OR        M00359	// LF_2D A¨¢A¡í AUAc ¨ú©ªA¨ö
LOADP     M00352	// LF_2D CODE READ
AND       M1902F	// DRY RUN
OR LOAD
OR        M19052	// LF_2D CODE SKIP
OR NOT    D003045.0	// LEFT 2D CODE USE
OR        M0035A	// LF_2D CODE OK
AND       M00357	// L_2D VC ON
AND NOT   M00852	// L_MES NG
OUT       M0035A	// LF_2D CODE OK
; L40
LOAD      M0035B	// LF_P&P 2D CODE OK PLS
AND<>     D003006 D000280	// 2D CODE 1ST CHARACTER / LF_1st CHARACTOR
AND<>     0 D003006	// 2D CODE 1ST CHARACTER
AND NOT   M1902F	// DRY RUN
AND NOT   M19052	// LF_2D CODE SKIP
AND       D003045.1	// 2D 2~5 ©ö©ªA¡Æ ©ö¢çAU¢¯¡© E¢çAI
OUT       M0035C	// LF_2D CODE CHARACTER NG
; L41
LOADP     M0035A	// LF_2D CODE OK
AND NOT   M0035D	// LF_2D A¨¢A¡í AUAc ¨ú©ªA¨ö KP
BMOV      D000200 D000280 h0008	// LF_2D CODE / LF_1st CHARACTOR
OUTP      M0035B	// LF_P&P 2D CODE OK PLS
; L43
LOADP     M00352	// LF_2D CODE READ
AND NOT   M01700	// Mes / Mes FileZilla
OUT       M00300	// LF_2D CODE START
; L44
LOADN     M00352	// LF_2D CODE READ
AND NOT   M01700	// Mes / Mes FileZilla
OUT       M00302	// LF_2D CODE STOP
// ======================== QR TIME ==========================
; L46
LOAD      M0035A	// LF_2D CODE OK
MOV       T1481 D019030	// L_QR TIME

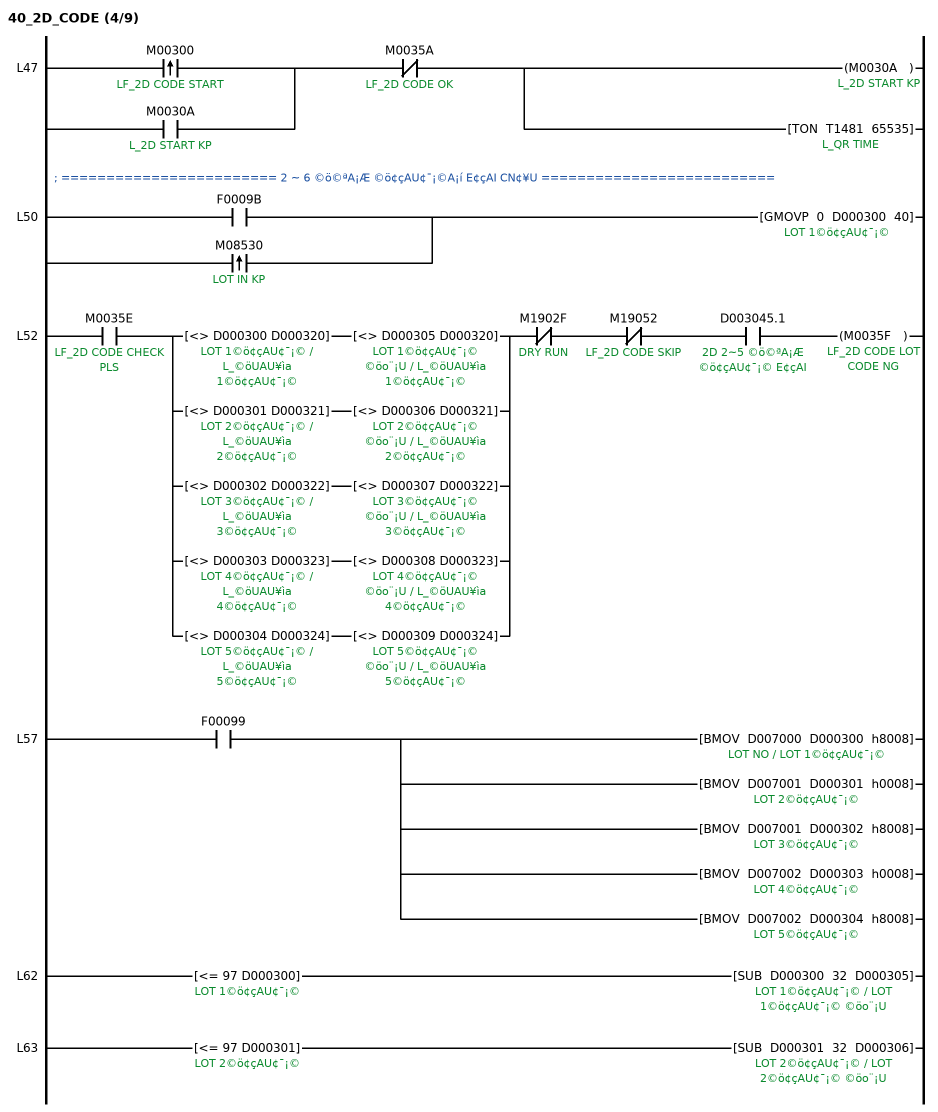
; L47
LOADP     M00300	// LF_2D CODE START
OR        M0030A	// L_2D START KP
AND NOT   M0035A	// LF_2D CODE OK
OUT       M0030A	// L_2D START KP
TON       T1481 65535	// L_QR TIME
// ======================== 2 ~ 6 ©ö©ªA¡Æ ©ö¢çAU¢¯¡©A¡í E¢çAI CN¢¥U ==========================
; L50
LOAD      F0009B
ORP       M08530	// LOT IN KP
GMOVP     0 D000300 40	// LOT 1©ö¢çAU¢¯¡©
; L52
LOAD      M0035E	// LF_2D CODE CHECK PLS
LOAD<>    D000300 D000320	// LOT 1©ö¢çAU¢¯¡© / L_©öUAU¥ìa 1©ö¢çAU¢¯¡©
AND<>     D000305 D000320	// LOT 1©ö¢çAU¢¯¡© ©öo¨¡U / L_©öUAU¥ìa 1©ö¢çAU¢¯¡©
LOAD<>    D000301 D000321	// LOT 2©ö¢çAU¢¯¡© / L_©öUAU¥ìa 2©ö¢çAU¢¯¡©
AND<>     D000306 D000321	// LOT 2©ö¢çAU¢¯¡© ©öo¨¡U / L_©öUAU¥ìa 2©ö¢çAU¢¯¡©
OR LOAD
LOAD<>    D000302 D000322	// LOT 3©ö¢çAU¢¯¡© / L_©öUAU¥ìa 3©ö¢çAU¢¯¡©
AND<>     D000307 D000322	// LOT 3©ö¢çAU¢¯¡© ©öo¨¡U / L_©öUAU¥ìa 3©ö¢çAU¢¯¡©
OR LOAD
LOAD<>    D000303 D000323	// LOT 4©ö¢çAU¢¯¡© / L_©öUAU¥ìa 4©ö¢çAU¢¯¡©
AND<>     D000308 D000323	// LOT 4©ö¢çAU¢¯¡© ©öo¨¡U / L_©öUAU¥ìa 4©ö¢çAU¢¯¡©
OR LOAD
LOAD<>    D000304 D000324	// LOT 5©ö¢çAU¢¯¡© / L_©öUAU¥ìa 5©ö¢çAU¢¯¡©
AND<>     D000309 D000324	// LOT 5©ö¢çAU¢¯¡© ©öo¨¡U / L_©öUAU¥ìa 5©ö¢çAU¢¯¡©
OR LOAD
AND LOAD
AND NOT   M1902F	// DRY RUN
AND NOT   M19052	// LF_2D CODE SKIP
AND       D003045.1	// 2D 2~5 ©ö©ªA¡Æ ©ö¢çAU¢¯¡© E¢çAI
OUT       M0035F	// LF_2D CODE LOT CODE NG
; L57
LOAD      F00099
BMOV      D007000 D000300 h8008	// LOT NO / LOT 1©ö¢çAU¢¯¡©
BMOV      D007001 D000301 h0008	// LOT 2©ö¢çAU¢¯¡©
BMOV      D007001 D000302 h8008	// LOT 3©ö¢çAU¢¯¡©
BMOV      D007002 D000303 h0008	// LOT 4©ö¢çAU¢¯¡©
BMOV      D007002 D000304 h8008	// LOT 5©ö¢çAU¢¯¡©
; L62
LOAD<=    97 D000300	// LOT 1©ö¢çAU¢¯¡©
SUB       D000300 32 D000305	// LOT 1©ö¢çAU¢¯¡© / LOT 1©ö¢çAU¢¯¡© ©öo¨¡U
; L63
LOAD<=    97 D000301	// LOT 2©ö¢çAU¢¯¡©
SUB       D000301 32 D000306	// LOT 2©ö¢çAU¢¯¡© / LOT 2©ö¢çAU¢¯¡© ©öo¨¡U

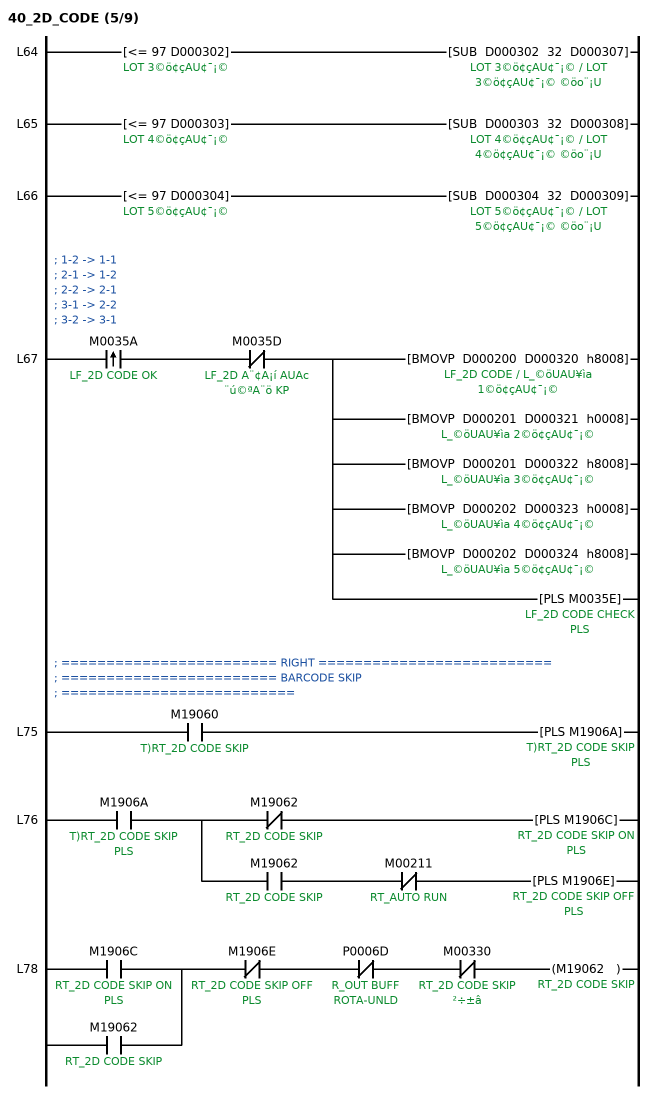
; L64
LOAD<=    97 D000302	// LOT 3©ö¢çAU¢¯¡©
SUB       D000302 32 D000307	// LOT 3©ö¢çAU¢¯¡© / LOT 3©ö¢çAU¢¯¡© ©öo¨¡U
; L65
LOAD<=    97 D000303	// LOT 4©ö¢çAU¢¯¡©
SUB       D000303 32 D000308	// LOT 4©ö¢çAU¢¯¡© / LOT 4©ö¢çAU¢¯¡© ©öo¨¡U
; L66
LOAD<=    97 D000304	// LOT 5©ö¢çAU¢¯¡©
SUB       D000304 32 D000309	// LOT 5©ö¢çAU¢¯¡© / LOT 5©ö¢çAU¢¯¡© ©öo¨¡U
; L67
LOADP     M0035A	// LF_2D CODE OK
AND NOT   M0035D	// LF_2D A¨¢A¡í AUAc ¨ú©ªA¨ö KP
BMOVP     D000200 D000320 h8008	// LF_2D CODE / L_©öUAU¥ìa 1©ö¢çAU¢¯¡©
BMOVP     D000201 D000321 h0008	// L_©öUAU¥ìa 2©ö¢çAU¢¯¡©
BMOVP     D000201 D000322 h8008	// L_©öUAU¥ìa 3©ö¢çAU¢¯¡©
BMOVP     D000202 D000323 h0008	// L_©öUAU¥ìa 4©ö¢çAU¢¯¡©
BMOVP     D000202 D000324 h8008	// L_©öUAU¥ìa 5©ö¢çAU¢¯¡©
OUTP      M0035E	// LF_2D CODE CHECK PLS
// output comment: 1-2 -> 1-1
// output comment: 2-1 -> 1-2
// output comment: 2-2 -> 2-1
// output comment: 3-1 -> 2-2
// output comment: 3-2 -> 3-1
// ======================== RIGHT ==========================
// ======================== BARCODE SKIP ==========================
; L75
LOAD      M19060	// T)RT_2D CODE SKIP
OUTP      M1906A	// T)RT_2D CODE SKIP PLS
; L76
LOAD      M1906A	// T)RT_2D CODE SKIP PLS
MPUSH
AND NOT   M19062	// RT_2D CODE SKIP
OUTP      M1906C	// RT_2D CODE SKIP ON PLS
MPOP
AND       M19062	// RT_2D CODE SKIP
AND NOT   M00211	// RT_AUTO RUN
OUTP      M1906E	// RT_2D CODE SKIP OFF PLS
; L78
LOAD      M1906C	// RT_2D CODE SKIP ON PLS
OR        M19062	// RT_2D CODE SKIP
AND NOT   M1906E	// RT_2D CODE SKIP OFF PLS
AND NOT   P0006D	// R_OUT BUFF ROTA-UNLD
AND NOT   M00330	// RT_2D CODE SKIP ²÷±â
OUT       M19062	// RT_2D CODE SKIP

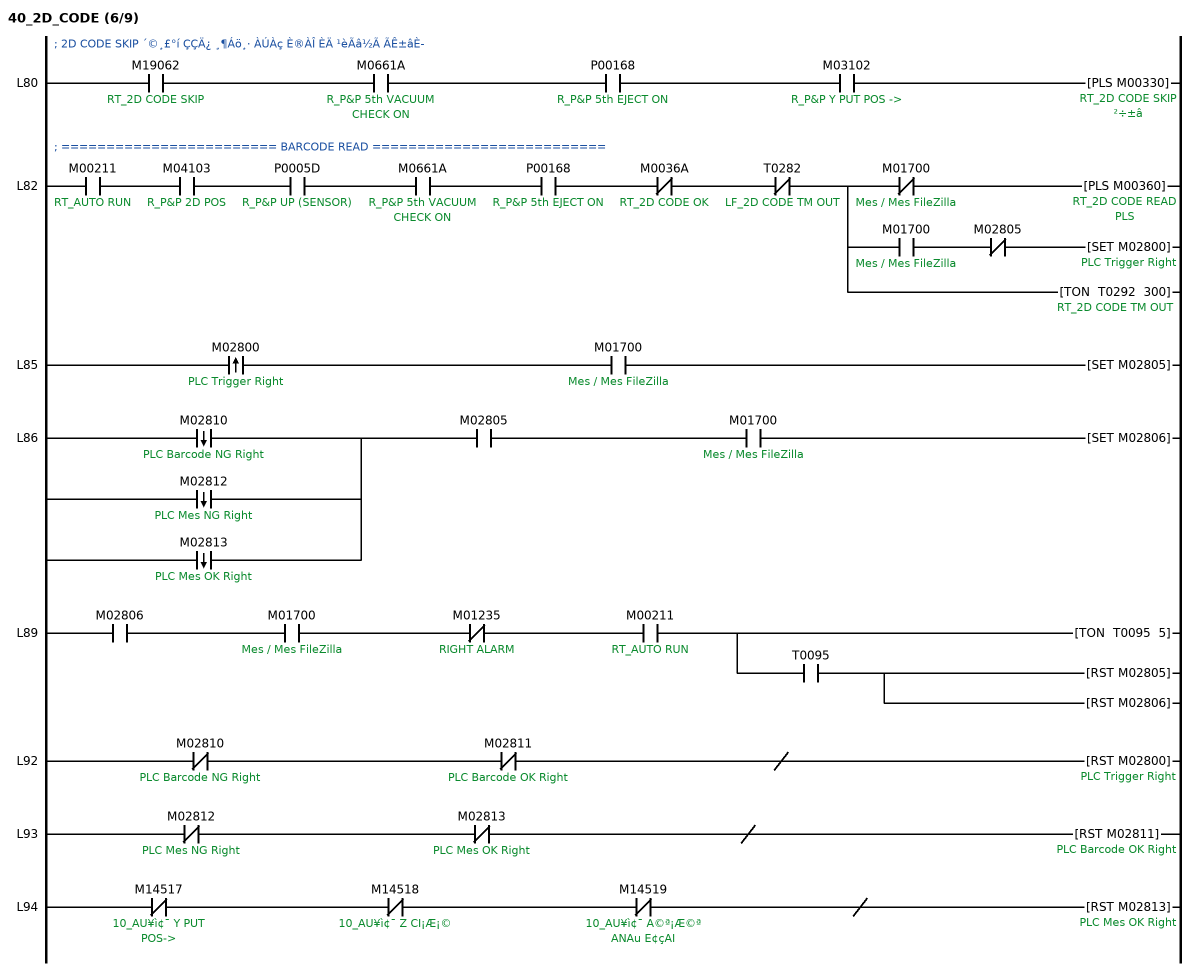
; L80
LOAD      M19062	// RT_2D CODE SKIP
AND       M0661A	// R_P&P 5th VACUUM CHECK ON
AND       P00168	// R_P&P 5th EJECT ON
AND       M03102	// R_P&P Y PUT POS ->
OUTP      M00330	// RT_2D CODE SKIP ²÷±â
// output comment: 2D CODE SKIP ´©¸£°í ÇÇÄ¿ ¸¶Áö¸· ÀÚÀç È®ÀÎ ÈÄ ¹èÃâ½Ã ÃÊ±âÈ­
// ======================== BARCODE READ ==========================
; L82
LOAD      M00211	// RT_AUTO RUN
AND       M04103	// R_P&P 2D POS
AND       P0005D	// R_P&P UP (SENSOR)
AND       M0661A	// R_P&P 5th VACUUM CHECK ON
AND       P00168	// R_P&P 5th EJECT ON
AND NOT   M0036A	// RT_2D CODE OK
AND NOT   T0282	// LF_2D CODE TM OUT
MPUSH
AND NOT   M01700	// Mes / Mes FileZilla
OUTP      M00360	// RT_2D CODE READ PLS
MLOAD
AND       M01700	// Mes / Mes FileZilla
AND NOT   M02805
SET       M02800	// PLC Trigger Right
MPOP
TON       T0292 300	// RT_2D CODE TM OUT
; L85
LOADP     M02800	// PLC Trigger Right
AND       M01700	// Mes / Mes FileZilla
SET       M02805
; L86
LOADN     M02810	// PLC Barcode NG Right
ORN       M02812	// PLC Mes NG Right
ORN       M02813	// PLC Mes OK Right
AND       M02805
AND       M01700	// Mes / Mes FileZilla
SET       M02806
; L89
LOAD      M02806
AND       M01700	// Mes / Mes FileZilla
AND NOT   M01235	// RIGHT ALARM
AND       M00211	// RT_AUTO RUN
TON       T0095 5
AND       T0095
RST       M02805
RST       M02806
; L92
LOAD NOT  M02810	// PLC Barcode NG Right
AND NOT   M02811	// PLC Barcode OK Right
NOT
RST       M02800	// PLC Trigger Right
; L93
LOAD NOT  M02812	// PLC Mes NG Right
AND NOT   M02813	// PLC Mes OK Right
NOT
RST       M02811	// PLC Barcode OK Right
; L94
LOAD NOT  M14517	// 10_AU¥ì¢¯ Y PUT POS->
AND NOT   M14518	// 10_AU¥ì¢¯ Z CI¡Æ¡©
AND NOT   M14519	// 10_AU¥ì¢¯ A©ª¡Æ©ª ANAu E¢çAI
NOT
RST       M02813	// PLC Mes OK Right

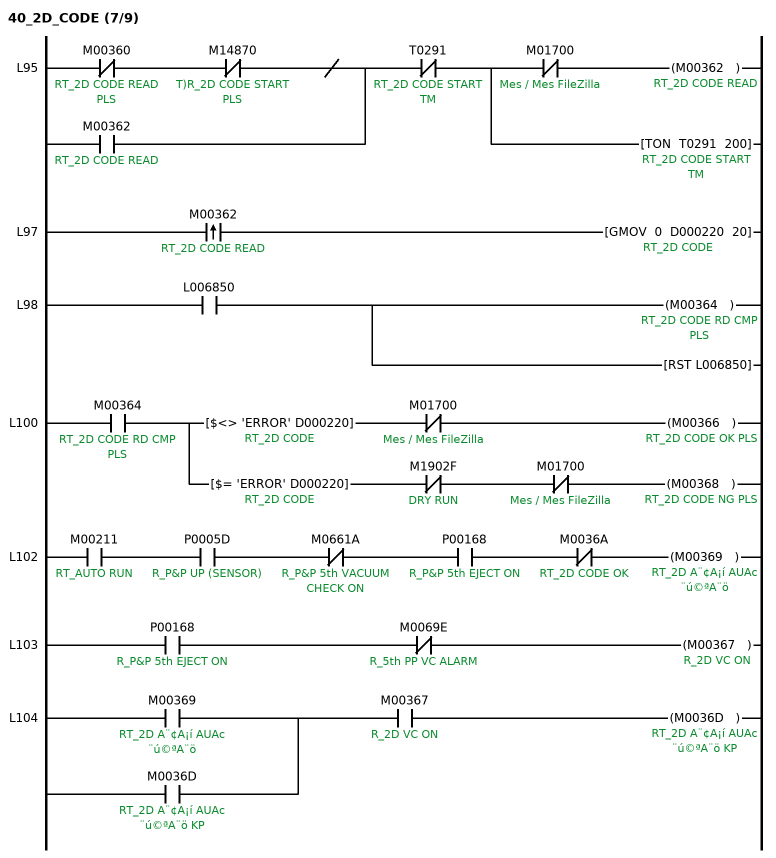
; L95
LOAD NOT  M00360	// RT_2D CODE READ PLS
AND NOT   M14870	// T)R_2D CODE START PLS
NOT
OR        M00362	// RT_2D CODE READ
AND NOT   T0291	// RT_2D CODE START TM
MPUSH
AND NOT   M01700	// Mes / Mes FileZilla
OUT       M00362	// RT_2D CODE READ
MPOP
TON       T0291 200	// RT_2D CODE START TM
; L97
LOADP     M00362	// RT_2D CODE READ
GMOV      0 D000220 20	// RT_2D CODE
; L98
LOAD      L006850
OUT       M00364	// RT_2D CODE RD CMP PLS
RST       L006850
; L100
LOAD      M00364	// RT_2D CODE RD CMP PLS
MPUSH
AND$<>    'ERROR' D000220	// RT_2D CODE
AND NOT   M01700	// Mes / Mes FileZilla
OUT       M00366	// RT_2D CODE OK PLS
MPOP
AND$=     'ERROR' D000220	// RT_2D CODE
AND NOT   M1902F	// DRY RUN
AND NOT   M01700	// Mes / Mes FileZilla
OUT       M00368	// RT_2D CODE NG PLS
; L102
LOAD      M00211	// RT_AUTO RUN
AND       P0005D	// R_P&P UP (SENSOR)
AND NOT   M0661A	// R_P&P 5th VACUUM CHECK ON
AND       P00168	// R_P&P 5th EJECT ON
AND NOT   M0036A	// RT_2D CODE OK
OUT       M00369	// RT_2D A¨¢A¡í AUAc ¨ú©ªA¨ö
; L103
LOAD      P00168	// R_P&P 5th EJECT ON
AND NOT   M0069E	// R_5th PP VC ALARM
OUT       M00367	// R_2D VC ON
; L104
LOAD      M00369	// RT_2D A¨¢A¡í AUAc ¨ú©ªA¨ö
OR        M0036D	// RT_2D A¨¢A¡í AUAc ¨ú©ªA¨ö KP
AND       M00367	// R_2D VC ON
OUT       M0036D	// RT_2D A¨¢A¡í AUAc ¨ú©ªA¨ö KP

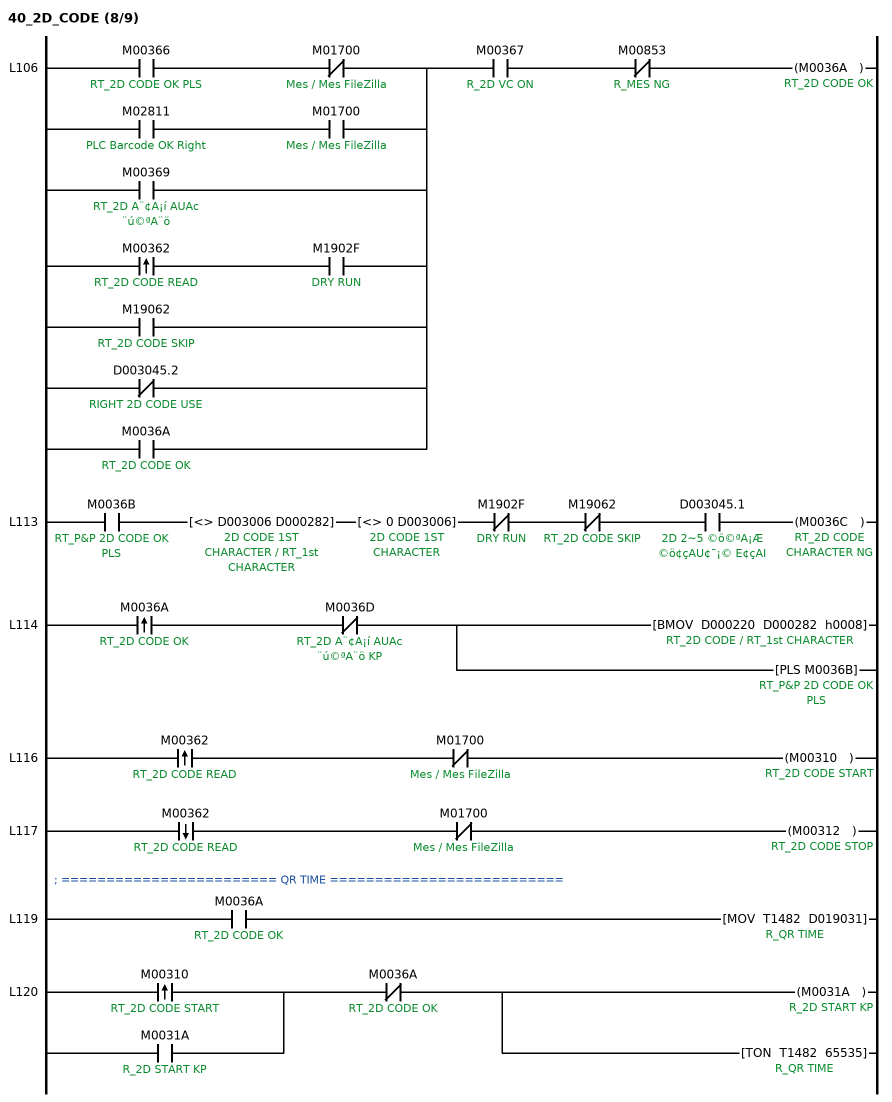
; L106
LOAD      M00366	// RT_2D CODE OK PLS
AND NOT   M01700	// Mes / Mes FileZilla
LOAD      M02811	// PLC Barcode OK Right
AND       M01700	// Mes / Mes FileZilla
OR LOAD
OR        M00369	// RT_2D A¨¢A¡í AUAc ¨ú©ªA¨ö
LOADP     M00362	// RT_2D CODE READ
AND       M1902F	// DRY RUN
OR LOAD
OR        M19062	// RT_2D CODE SKIP
OR NOT    D003045.2	// RIGHT 2D CODE USE
OR        M0036A	// RT_2D CODE OK
AND       M00367	// R_2D VC ON
AND NOT   M00853	// R_MES NG
OUT       M0036A	// RT_2D CODE OK
; L113
LOAD      M0036B	// RT_P&P 2D CODE OK PLS
AND<>     D003006 D000282	// 2D CODE 1ST CHARACTER / RT_1st CHARACTER
AND<>     0 D003006	// 2D CODE 1ST CHARACTER
AND NOT   M1902F	// DRY RUN
AND NOT   M19062	// RT_2D CODE SKIP
AND       D003045.1	// 2D 2~5 ©ö©ªA¡Æ ©ö¢çAU¢¯¡© E¢çAI
OUT       M0036C	// RT_2D CODE CHARACTER NG
; L114
LOADP     M0036A	// RT_2D CODE OK
AND NOT   M0036D	// RT_2D A¨¢A¡í AUAc ¨ú©ªA¨ö KP
BMOV      D000220 D000282 h0008	// RT_2D CODE / RT_1st CHARACTER
OUTP      M0036B	// RT_P&P 2D CODE OK PLS
; L116
LOADP     M00362	// RT_2D CODE READ
AND NOT   M01700	// Mes / Mes FileZilla
OUT       M00310	// RT_2D CODE START
; L117
LOADN     M00362	// RT_2D CODE READ
AND NOT   M01700	// Mes / Mes FileZilla
OUT       M00312	// RT_2D CODE STOP
// ======================== QR TIME ==========================
; L119
LOAD      M0036A	// RT_2D CODE OK
MOV       T1482 D019031	// R_QR TIME
; L120
LOADP     M00310	// RT_2D CODE START
OR        M0031A	// R_2D START KP
AND NOT   M0036A	// RT_2D CODE OK
OUT       M0031A	// R_2D START KP
TON       T1482 65535	// R_QR TIME

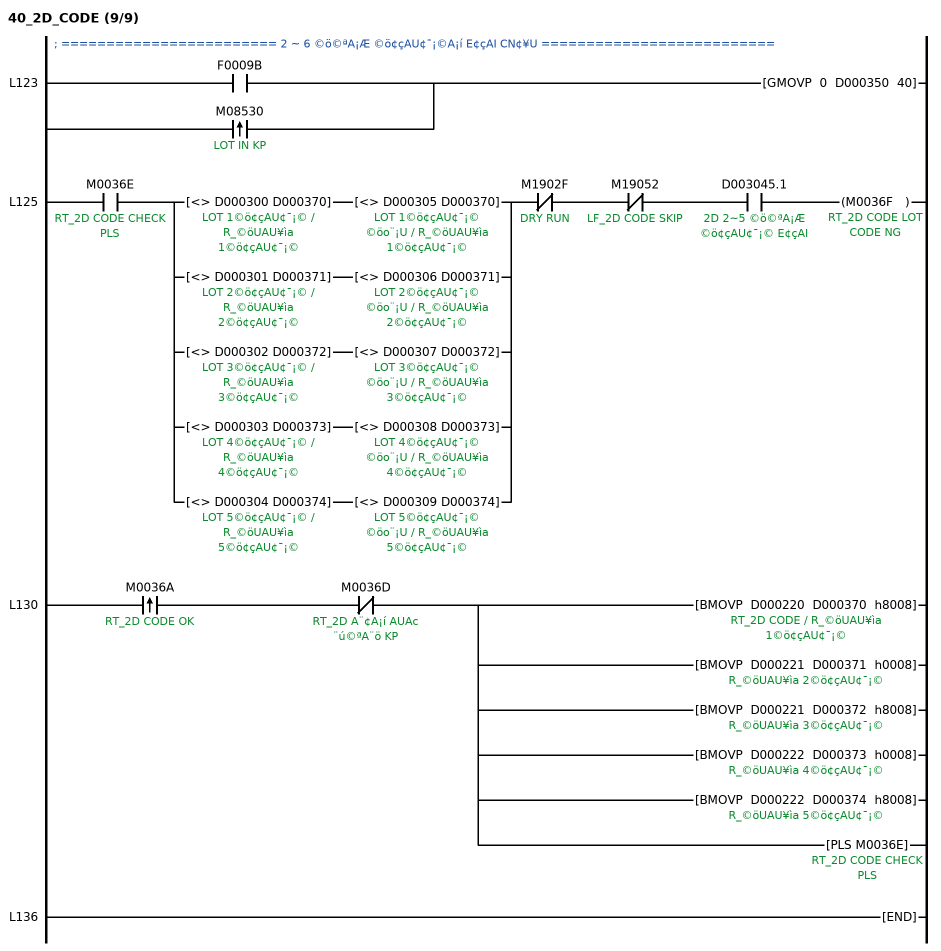
// ======================== 2 ~ 6 ©ö©ªA¡Æ ©ö¢çAU¢¯¡©A¡í E¢çAI CN¢¥U ==========================
; L123
LOAD      F0009B
ORP       M08530	// LOT IN KP
GMOVP     0 D000350 40
; L125
LOAD      M0036E	// RT_2D CODE CHECK PLS
LOAD<>    D000300 D000370	// LOT 1©ö¢çAU¢¯¡© / R_©öUAU¥ìa 1©ö¢çAU¢¯¡©
AND<>     D000305 D000370	// LOT 1©ö¢çAU¢¯¡© ©öo¨¡U / R_©öUAU¥ìa 1©ö¢çAU¢¯¡©
LOAD<>    D000301 D000371	// LOT 2©ö¢çAU¢¯¡© / R_©öUAU¥ìa 2©ö¢çAU¢¯¡©
AND<>     D000306 D000371	// LOT 2©ö¢çAU¢¯¡© ©öo¨¡U / R_©öUAU¥ìa 2©ö¢çAU¢¯¡©
OR LOAD
LOAD<>    D000302 D000372	// LOT 3©ö¢çAU¢¯¡© / R_©öUAU¥ìa 3©ö¢çAU¢¯¡©
AND<>     D000307 D000372	// LOT 3©ö¢çAU¢¯¡© ©öo¨¡U / R_©öUAU¥ìa 3©ö¢çAU¢¯¡©
OR LOAD
LOAD<>    D000303 D000373	// LOT 4©ö¢çAU¢¯¡© / R_©öUAU¥ìa 4©ö¢çAU¢¯¡©
AND<>     D000308 D000373	// LOT 4©ö¢çAU¢¯¡© ©öo¨¡U / R_©öUAU¥ìa 4©ö¢çAU¢¯¡©
OR LOAD
LOAD<>    D000304 D000374	// LOT 5©ö¢çAU¢¯¡© / R_©öUAU¥ìa 5©ö¢çAU¢¯¡©
AND<>     D000309 D000374	// LOT 5©ö¢çAU¢¯¡© ©öo¨¡U / R_©öUAU¥ìa 5©ö¢çAU¢¯¡©
OR LOAD
AND LOAD
AND NOT   M1902F	// DRY RUN
AND NOT   M19052	// LF_2D CODE SKIP
AND       D003045.1	// 2D 2~5 ©ö©ªA¡Æ ©ö¢çAU¢¯¡© E¢çAI
OUT       M0036F	// RT_2D CODE LOT CODE NG
; L130
LOADP     M0036A	// RT_2D CODE OK
AND NOT   M0036D	// RT_2D A¨¢A¡í AUAc ¨ú©ªA¨ö KP
BMOVP     D000220 D000370 h8008	// RT_2D CODE / R_©öUAU¥ìa 1©ö¢çAU¢¯¡©
BMOVP     D000221 D000371 h0008	// R_©öUAU¥ìa 2©ö¢çAU¢¯¡©
BMOVP     D000221 D000372 h8008	// R_©öUAU¥ìa 3©ö¢çAU¢¯¡©
BMOVP     D000222 D000373 h0008	// R_©öUAU¥ìa 4©ö¢çAU¢¯¡©
BMOVP     D000222 D000374 h8008	// R_©öUAU¥ìa 5©ö¢çAU¢¯¡©
OUTP      M0036E	// RT_2D CODE CHECK PLS
; L136
END

PROGRAM 41_MES (task: ¨ö¨¬A¥ì CA¡¤I¡¾¡¿¡¤¡Í)

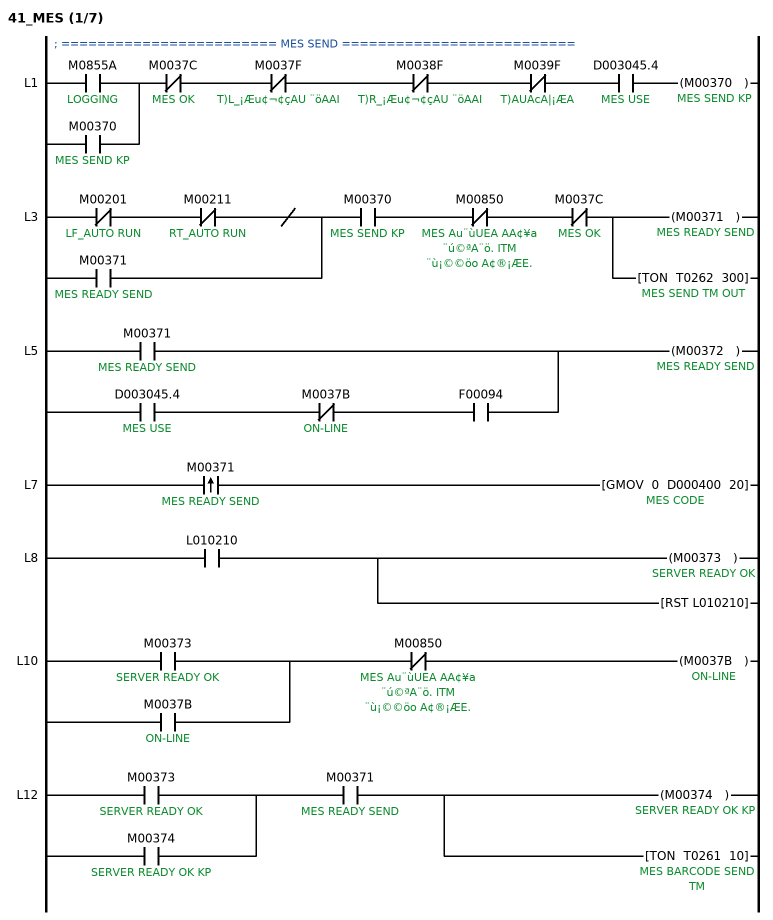
// ======================== MES SEND ==========================
; L1
LOAD      M0855A	// LOGGING
OR        M00370	// MES SEND KP
AND NOT   M0037C	// MES OK
AND NOT   M0037F	// T)L_¡Æu¢¬¢çAU ¨öAAI
AND NOT   M0038F	// T)R_¡Æu¢¬¢çAU ¨öAAI
AND NOT   M0039F	// T)AUAcA|¡ÆA
AND       D003045.4	// MES USE
OUT       M00370	// MES SEND KP
; L3
LOAD NOT  M00201	// LF_AUTO RUN
AND NOT   M00211	// RT_AUTO RUN
NOT
OR        M00371	// MES READY SEND
AND       M00370	// MES SEND KP
AND NOT   M00850	// MES Au¨ùUEA AA¢¥a ¨ú©ªA¨ö. ITM ¨ù¡©©öo A¢®¡ÆE.
AND NOT   M0037C	// MES OK
OUT       M00371	// MES READY SEND
TON       T0262 300	// MES SEND TM OUT
; L5
LOAD      M00371	// MES READY SEND
LOAD      D003045.4	// MES USE
AND NOT   M0037B	// ON-LINE
AND       F00094
OR LOAD
OUT       M00372	// MES READY SEND
; L7
LOADP     M00371	// MES READY SEND
GMOV      0 D000400 20	// MES CODE
; L8
LOAD      L010210
OUT       M00373	// SERVER READY OK
RST       L010210
; L10
LOAD      M00373	// SERVER READY OK
OR        M0037B	// ON-LINE
AND NOT   M00850	// MES Au¨ùUEA AA¢¥a ¨ú©ªA¨ö. ITM ¨ù¡©©öo A¢®¡ÆE.
OUT       M0037B	// ON-LINE
; L12
LOAD      M00373	// SERVER READY OK
OR        M00374	// SERVER READY OK KP
AND       M00371	// MES READY SEND
OUT       M00374	// SERVER READY OK KP
TON       T0261 10	// MES BARCODE SEND TM

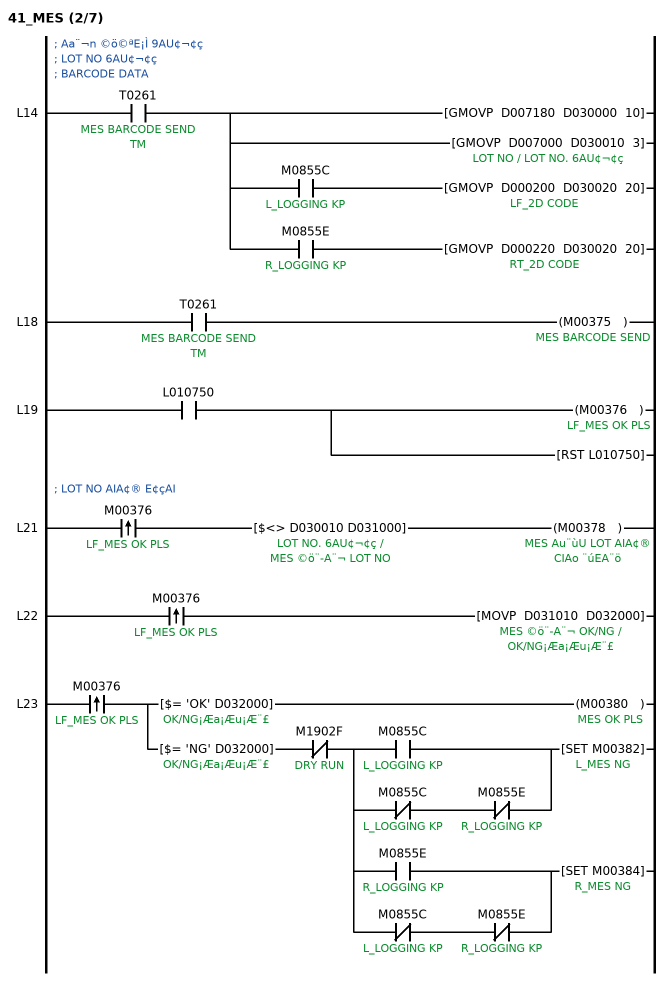
; L14
LOAD      T0261	// MES BARCODE SEND TM
GMOVP     D007180 D030000 10
GMOVP     D007000 D030010 3	// LOT NO / LOT NO. 6AU¢¬¢ç
MPUSH
AND       M0855C	// L_LOGGING KP
GMOVP     D000200 D030020 20	// LF_2D CODE
MPOP
AND       M0855E	// R_LOGGING KP
GMOVP     D000220 D030020 20	// RT_2D CODE
// output comment: Aa¨¬n ©ö©ªE¡Ì 9AU¢¬¢ç
// output comment: LOT NO 6AU¢¬¢ç
// output comment: BARCODE DATA
; L18
LOAD      T0261	// MES BARCODE SEND TM
OUT       M00375	// MES BARCODE SEND
; L19
LOAD      L010750
OUT       M00376	// LF_MES OK PLS
RST       L010750
; L21
LOADP     M00376	// LF_MES OK PLS
AND$<>    D030010 D031000	// LOT NO. 6AU¢¬¢ç / MES ©ö¨­A¨¬ LOT NO
OUT       M00378	// MES Au¨ùU LOT AIA¢® CIAo ¨úEA¨ö
// output comment: LOT NO AIA¢® E¢çAI
; L22
LOADP     M00376	// LF_MES OK PLS
MOVP      D031010 D032000	// MES ©ö¨­A¨¬ OK/NG / OK/NG¡Æa¡Æu¡Æ¨£
; L23
LOADP     M00376	// LF_MES OK PLS
MPUSH
AND$=     'OK' D032000	// OK/NG¡Æa¡Æu¡Æ¨£
OUT       M00380	// MES OK PLS
MPOP
AND$=     'NG' D032000	// OK/NG¡Æa¡Æu¡Æ¨£
AND NOT   M1902F	// DRY RUN
MPUSH
LOAD      M0855C	// L_LOGGING KP
LOAD NOT  M0855C	// L_LOGGING KP
AND NOT   M0855E	// R_LOGGING KP
OR LOAD
AND LOAD
SET       M00382	// L_MES NG
MPOP
LOAD      M0855E	// R_LOGGING KP
LOAD NOT  M0855C	// L_LOGGING KP
AND NOT   M0855E	// R_LOGGING KP
OR LOAD
AND LOAD
SET       M00384	// R_MES NG

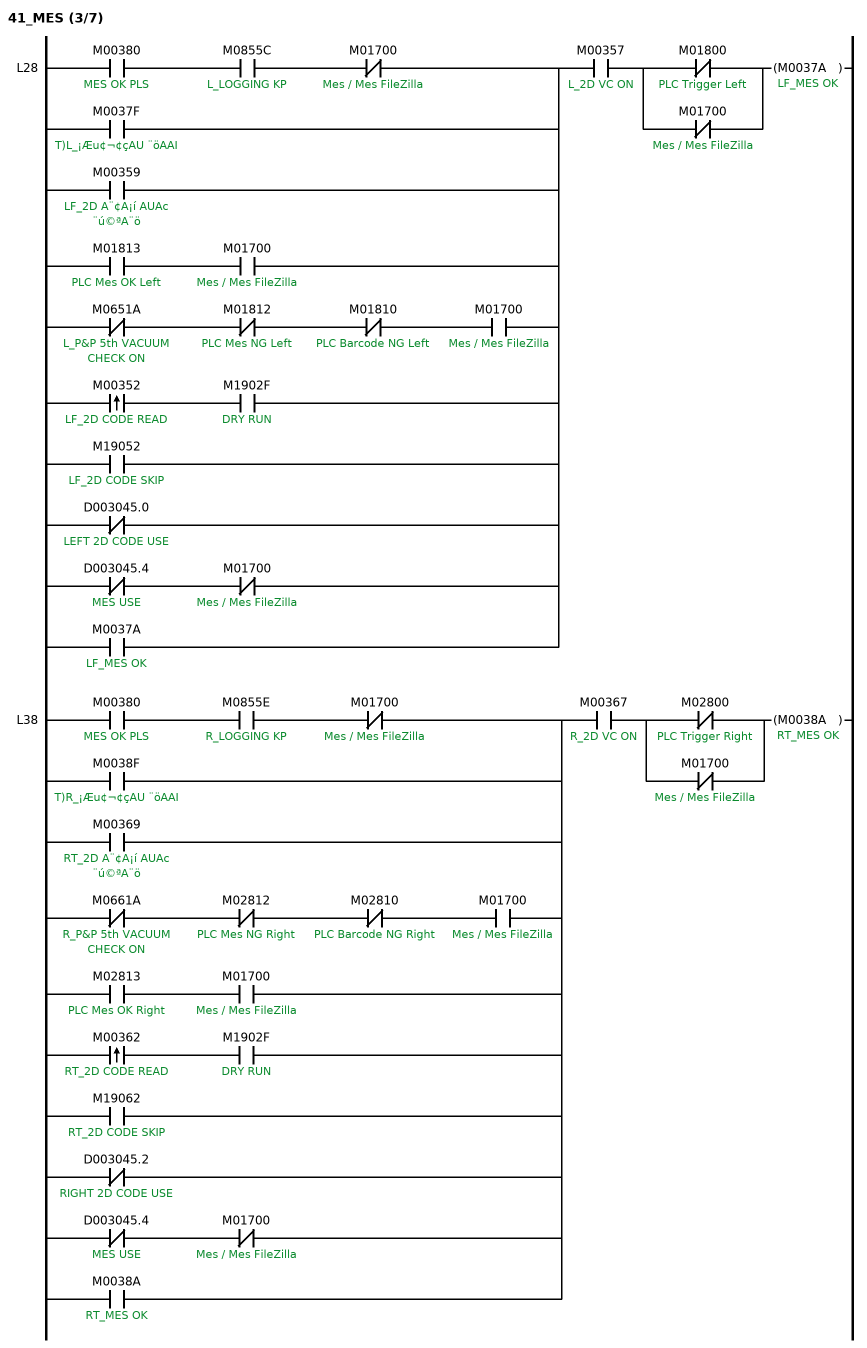
; L28
LOAD      M00380	// MES OK PLS
AND       M0855C	// L_LOGGING KP
AND NOT   M01700	// Mes / Mes FileZilla
OR        M0037F	// T)L_¡Æu¢¬¢çAU ¨öAAI
OR        M00359	// LF_2D A¨¢A¡í AUAc ¨ú©ªA¨ö
LOAD      M01813	// PLC Mes OK Left
AND       M01700	// Mes / Mes FileZilla
OR LOAD
LOAD NOT  M0651A	// L_P&P 5th VACUUM CHECK ON
AND NOT   M01812	// PLC Mes NG Left
AND NOT   M01810	// PLC Barcode NG Left
AND       M01700	// Mes / Mes FileZilla
OR LOAD
LOADP     M00352	// LF_2D CODE READ
AND       M1902F	// DRY RUN
OR LOAD
OR        M19052	// LF_2D CODE SKIP
OR NOT    D003045.0	// LEFT 2D CODE USE
LOAD NOT  D003045.4	// MES USE
AND NOT   M01700	// Mes / Mes FileZilla
OR LOAD
OR        M0037A	// LF_MES OK
AND       M00357	// L_2D VC ON
LOAD NOT  M01800	// PLC Trigger Left
OR NOT    M01700	// Mes / Mes FileZilla
AND LOAD
OUT       M0037A	// LF_MES OK
; L38
LOAD      M00380	// MES OK PLS
AND       M0855E	// R_LOGGING KP
AND NOT   M01700	// Mes / Mes FileZilla
OR        M0038F	// T)R_¡Æu¢¬¢çAU ¨öAAI
OR        M00369	// RT_2D A¨¢A¡í AUAc ¨ú©ªA¨ö
LOAD NOT  M0661A	// R_P&P 5th VACUUM CHECK ON
AND NOT   M02812	// PLC Mes NG Right
AND NOT   M02810	// PLC Barcode NG Right
AND       M01700	// Mes / Mes FileZilla
OR LOAD
LOAD      M02813	// PLC Mes OK Right
AND       M01700	// Mes / Mes FileZilla
OR LOAD
LOADP     M00362	// RT_2D CODE READ
AND       M1902F	// DRY RUN
OR LOAD
OR        M19062	// RT_2D CODE SKIP
OR NOT    D003045.2	// RIGHT 2D CODE USE
LOAD NOT  D003045.4	// MES USE
AND NOT   M01700	// Mes / Mes FileZilla
OR LOAD
OR        M0038A	// RT_MES OK
AND       M00367	// R_2D VC ON
LOAD NOT  M02800	// PLC Trigger Right
OR NOT    M01700	// Mes / Mes FileZilla
AND LOAD
OUT       M0038A	// RT_MES OK

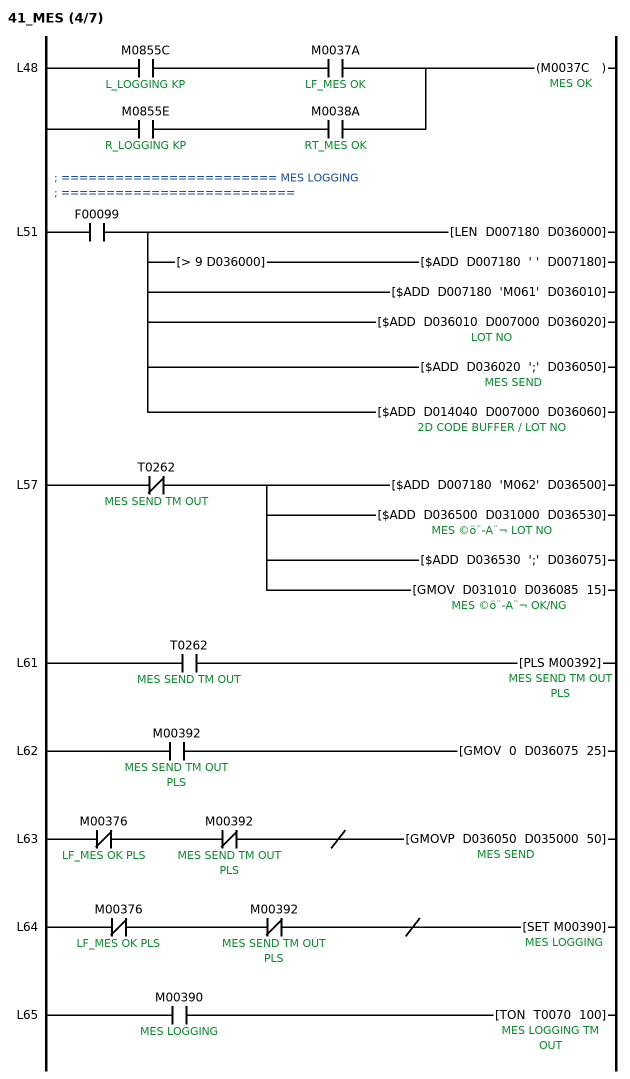
; L48
LOAD      M0855C	// L_LOGGING KP
AND       M0037A	// LF_MES OK
LOAD      M0855E	// R_LOGGING KP
AND       M0038A	// RT_MES OK
OR LOAD
OUT       M0037C	// MES OK
// ======================== MES LOGGING ==========================
; L51
LOAD      F00099
LEN       D007180 D036000
MPUSH
AND>      9 D036000
$ADD      D007180 ' ' D007180
MPOP
$ADD      D007180 'M061' D036010
$ADD      D036010 D007000 D036020	// LOT NO
$ADD      D036020 ';' D036050	// MES SEND
$ADD      D014040 D007000 D036060	// 2D CODE BUFFER / LOT NO
; L57
LOAD NOT  T0262	// MES SEND TM OUT
$ADD      D007180 'M062' D036500
$ADD      D036500 D031000 D036530	// MES ©ö¨­A¨¬ LOT NO
$ADD      D036530 ';' D036075
GMOV      D031010 D036085 15	// MES ©ö¨­A¨¬ OK/NG
; L61
LOAD      T0262	// MES SEND TM OUT
OUTP      M00392	// MES SEND TM OUT PLS
; L62
LOAD      M00392	// MES SEND TM OUT PLS
GMOV      0 D036075 25
; L63
LOAD NOT  M00376	// LF_MES OK PLS
AND NOT   M00392	// MES SEND TM OUT PLS
NOT
GMOVP     D036050 D035000 50	// MES SEND
; L64
LOAD NOT  M00376	// LF_MES OK PLS
AND NOT   M00392	// MES SEND TM OUT PLS
NOT
SET       M00390	// MES LOGGING
; L65
LOAD      M00390	// MES LOGGING
TON       T0070 100	// MES LOGGING TM OUT

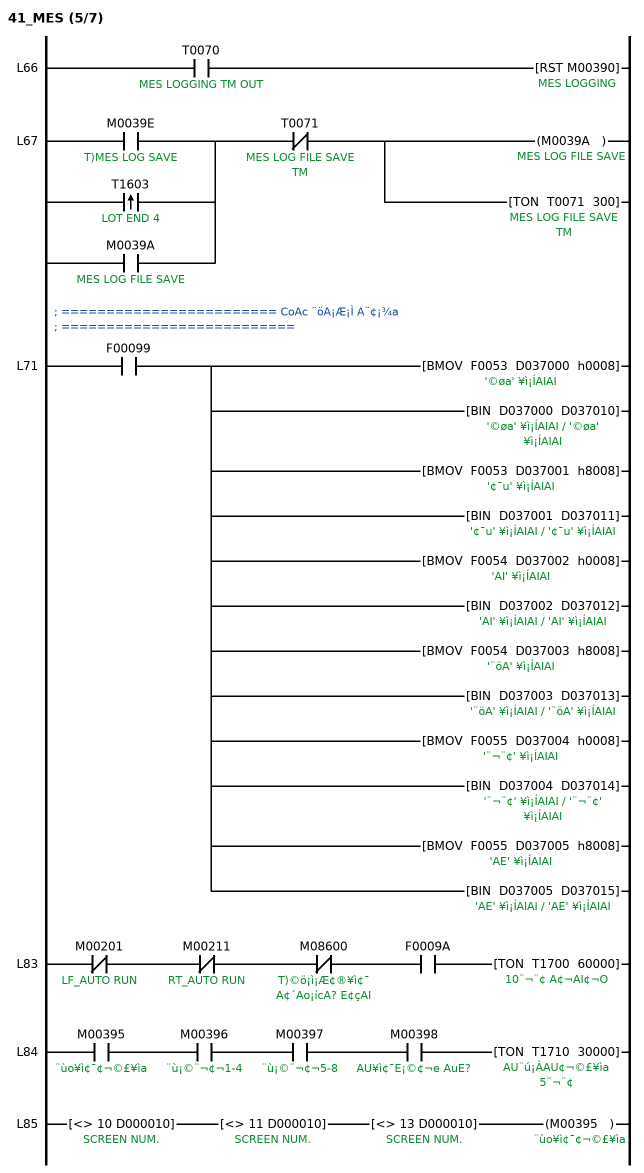
; L66
LOAD      T0070	// MES LOGGING TM OUT
RST       M00390	// MES LOGGING
; L67
LOAD      M0039E	// T)MES LOG SAVE
ORP       T1603	// LOT END 4
OR        M0039A	// MES LOG FILE SAVE
AND NOT   T0071	// MES LOG FILE SAVE TM
OUT       M0039A	// MES LOG FILE SAVE
TON       T0071 300	// MES LOG FILE SAVE TM
// ======================== CoAc ¨öA¡Æ¡Ì A¨¢¡¾a ==========================
; L71
LOAD      F00099
BMOV      F0053 D037000 h0008	// '©øa' ¥ì¡ÍAIAI
BIN       D037000 D037010	// '©øa' ¥ì¡ÍAIAI / '©øa' ¥ì¡ÍAIAI
BMOV      F0053 D037001 h8008	// '¢¯u' ¥ì¡ÍAIAI
BIN       D037001 D037011	// '¢¯u' ¥ì¡ÍAIAI / '¢¯u' ¥ì¡ÍAIAI
BMOV      F0054 D037002 h0008	// 'AI' ¥ì¡ÍAIAI
BIN       D037002 D037012	// 'AI' ¥ì¡ÍAIAI / 'AI' ¥ì¡ÍAIAI
BMOV      F0054 D037003 h8008	// '¨öA' ¥ì¡ÍAIAI
BIN       D037003 D037013	// '¨öA' ¥ì¡ÍAIAI / '¨öA' ¥ì¡ÍAIAI
BMOV      F0055 D037004 h0008	// '¨¬¨¢' ¥ì¡ÍAIAI
BIN       D037004 D037014	// '¨¬¨¢' ¥ì¡ÍAIAI / '¨¬¨¢' ¥ì¡ÍAIAI
BMOV      F0055 D037005 h8008	// 'AE' ¥ì¡ÍAIAI
BIN       D037005 D037015	// 'AE' ¥ì¡ÍAIAI / 'AE' ¥ì¡ÍAIAI
; L83
LOAD NOT  M00201	// LF_AUTO RUN
AND NOT   M00211	// RT_AUTO RUN
AND NOT   M08600	// T)©ö¡ì¡Æ¢®¥ì¢¯ A¢´Ao¡ícA? E¢çAI
AND       F0009A
TON       T1700 60000	// 10¨¬¨¢ A¢¬AI¢¬O
; L84
LOAD      M00395	// ¨ùo¥ì¢¯¢¬©£¥ìa
AND       M00396	// ¨ù¡©¨¬¢¬1-4
AND       M00397	// ¨ù¡©¨¬¢¬5-8
AND       M00398	// AU¥ì¢¯E¡©¢¬e AuE?
TON       T1710 30000	// AU¨ú¡ÀAU¢¬©£¥ìa 5¨¬¨¢
; L85
LOAD<>    10 D000010	// SCREEN NUM.
AND<>     11 D000010	// SCREEN NUM.
AND<>     13 D000010	// SCREEN NUM.
OUT       M00395	// ¨ùo¥ì¢¯¢¬©£¥ìa

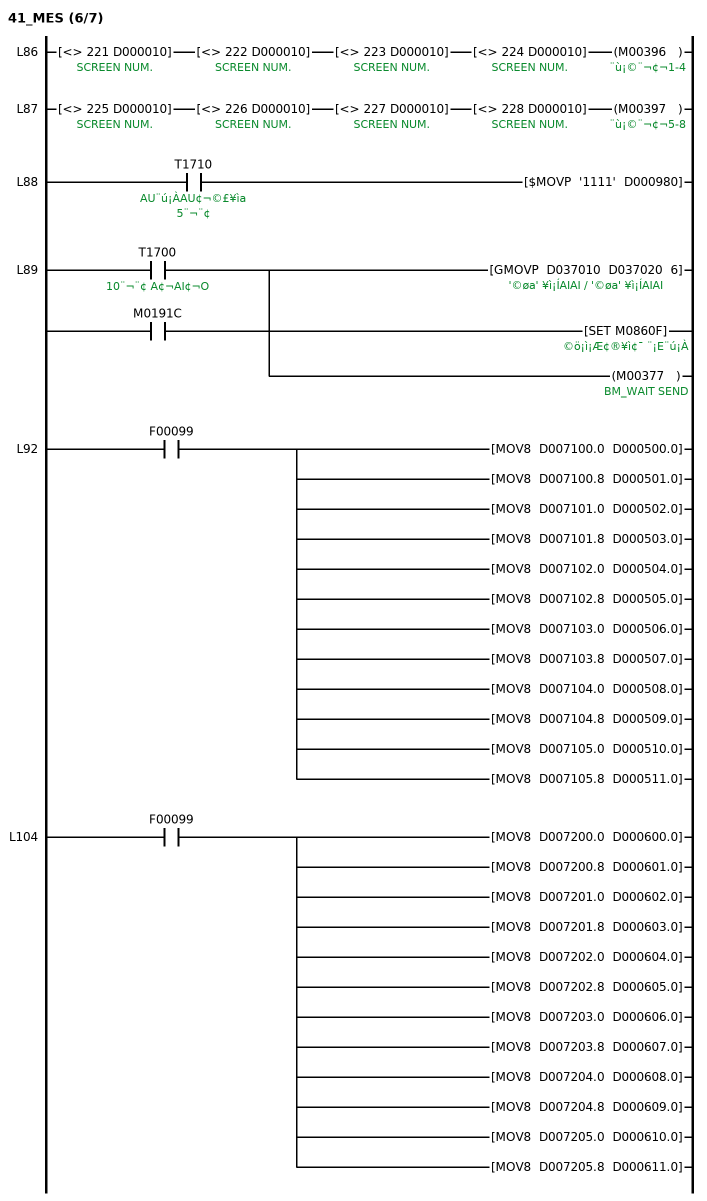
; L86
LOAD<>    221 D000010	// SCREEN NUM.
AND<>     222 D000010	// SCREEN NUM.
AND<>     223 D000010	// SCREEN NUM.
AND<>     224 D000010	// SCREEN NUM.
OUT       M00396	// ¨ù¡©¨¬¢¬1-4
; L87
LOAD<>    225 D000010	// SCREEN NUM.
AND<>     226 D000010	// SCREEN NUM.
AND<>     227 D000010	// SCREEN NUM.
AND<>     228 D000010	// SCREEN NUM.
OUT       M00397	// ¨ù¡©¨¬¢¬5-8
; L88
LOAD      T1710	// AU¨ú¡ÀAU¢¬©£¥ìa 5¨¬¨¢
$MOVP     '1111' D000980
; L89
LOAD      T1700	// 10¨¬¨¢ A¢¬AI¢¬O
OR        M0191C
GMOVP     D037010 D037020 6	// '©øa' ¥ì¡ÍAIAI / '©øa' ¥ì¡ÍAIAI
SET       M0860F	// ©ö¡ì¡Æ¢®¥ì¢¯ ¨¡E¨ú¡À
OUT       M00377	// BM_WAIT SEND
; L92
LOAD      F00099
MOV8      D007100.0 D000500.0
MOV8      D007100.8 D000501.0
MOV8      D007101.0 D000502.0
MOV8      D007101.8 D000503.0
MOV8      D007102.0 D000504.0
MOV8      D007102.8 D000505.0
MOV8      D007103.0 D000506.0
MOV8      D007103.8 D000507.0
MOV8      D007104.0 D000508.0
MOV8      D007104.8 D000509.0
MOV8      D007105.0 D000510.0
MOV8      D007105.8 D000511.0
; L104
LOAD      F00099
MOV8      D007200.0 D000600.0
MOV8      D007200.8 D000601.0
MOV8      D007201.0 D000602.0
MOV8      D007201.8 D000603.0
MOV8      D007202.0 D000604.0
MOV8      D007202.8 D000605.0
MOV8      D007203.0 D000606.0
MOV8      D007203.8 D000607.0
MOV8      D007204.0 D000608.0
MOV8      D007204.8 D000609.0
MOV8      D007205.0 D000610.0
MOV8      D007205.8 D000611.0

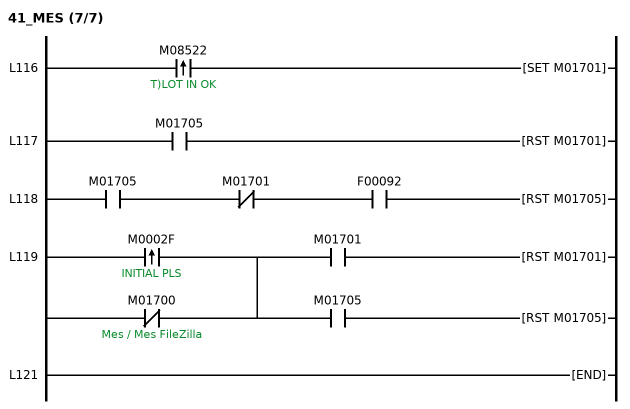
; L116
LOADP     M08522	// T)LOT IN OK
SET       M01701
; L117
LOAD      M01705
RST       M01701
; L118
LOAD      M01705
AND NOT   M01701
AND       F00092
RST       M01705
; L119
LOADP     M0002F	// INITIAL PLS
OR NOT    M01700	// Mes / Mes FileZilla
MPUSH
AND       M01701
RST       M01701
MPOP
AND       M01705
RST       M01705
; L121
END

PROGRAM 51_MT_01_2_3_4 (task: ¨ö¨¬A¥ì CA¡¤I¡¾¡¿¡¤¡Í)

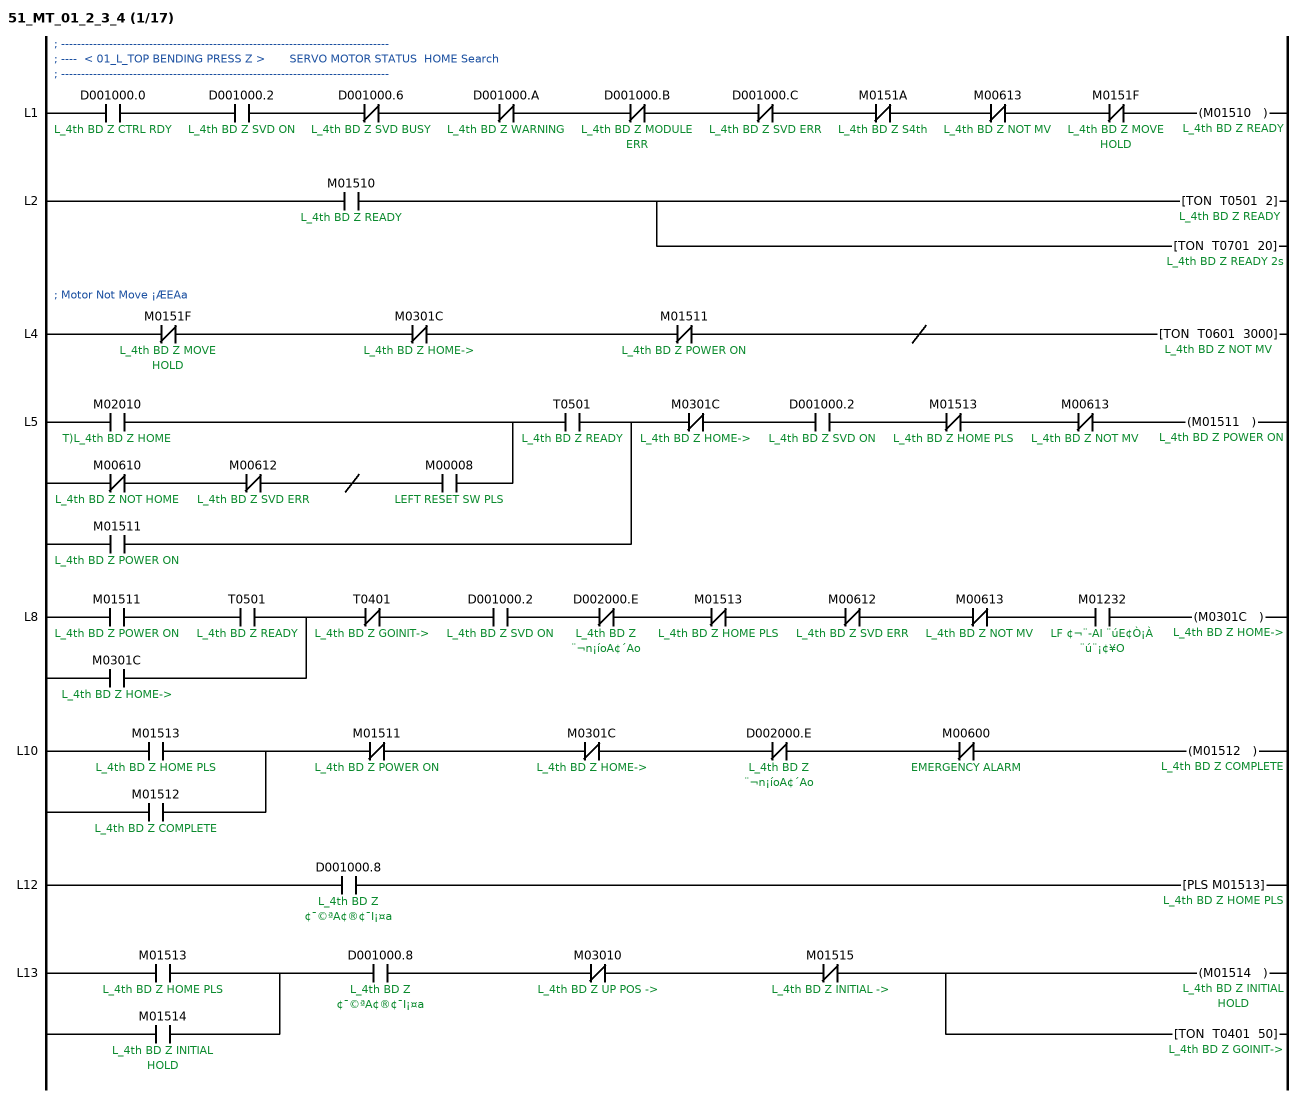
// ----------------------------------------------------------------------------------
// 
// ----  < 01_L_TOP BENDING PRESS Z >       SERVO MOTOR STATUS  HOME Search
// 
// ----------------------------------------------------------------------------------
; L1
LOAD      D001000.0	// L_4th BD Z CTRL RDY
AND       D001000.2	// L_4th BD Z SVD ON
AND NOT   D001000.6	// L_4th BD Z SVD BUSY
AND NOT   D001000.A	// L_4th BD Z WARNING
AND NOT   D001000.B	// L_4th BD Z MODULE ERR
AND NOT   D001000.C	// L_4th BD Z SVD ERR
AND NOT   M0151A	// L_4th BD Z S4th
AND NOT   M00613	// L_4th BD Z NOT MV
AND NOT   M0151F	// L_4th BD Z MOVE HOLD
OUT       M01510	// L_4th BD Z READY
; L2
LOAD      M01510	// L_4th BD Z READY
TON       T0501 2	// L_4th BD Z READY
TON       T0701 20	// L_4th BD Z READY 2s
; L4
LOAD NOT  M0151F	// L_4th BD Z MOVE HOLD
AND NOT   M0301C	// L_4th BD Z HOME->
AND NOT   M01511	// L_4th BD Z POWER ON
NOT
TON       T0601 3000	// L_4th BD Z NOT MV
// output comment: Motor Not Move ¡ÆEAa
; L5
LOAD      M02010	// T)L_4th BD Z HOME
LOAD NOT  M00610	// L_4th BD Z NOT HOME
AND NOT   M00612	// L_4th BD Z SVD ERR
NOT
AND       M00008	// LEFT RESET SW PLS
OR LOAD
AND       T0501	// L_4th BD Z READY
OR        M01511	// L_4th BD Z POWER ON
AND NOT   M0301C	// L_4th BD Z HOME->
AND       D001000.2	// L_4th BD Z SVD ON
AND NOT   M01513	// L_4th BD Z HOME PLS
AND NOT   M00613	// L_4th BD Z NOT MV
OUT       M01511	// L_4th BD Z POWER ON
; L8
LOAD      M01511	// L_4th BD Z POWER ON
AND       T0501	// L_4th BD Z READY
OR        M0301C	// L_4th BD Z HOME->
AND NOT   T0401	// L_4th BD Z GOINIT->
AND       D001000.2	// L_4th BD Z SVD ON
AND NOT   D002000.E	// L_4th BD Z ¨¬n¡íoA¢´Ao
AND NOT   M01513	// L_4th BD Z HOME PLS
AND NOT   M00612	// L_4th BD Z SVD ERR
AND NOT   M00613	// L_4th BD Z NOT MV
AND       M01232	// LF ¢¬¨­AI ¨úE¢Ò¡À ¨ú¨¡¢¥O
OUT       M0301C	// L_4th BD Z HOME->
; L10
LOAD      M01513	// L_4th BD Z HOME PLS
OR        M01512	// L_4th BD Z COMPLETE
AND NOT   M01511	// L_4th BD Z POWER ON
AND NOT   M0301C	// L_4th BD Z HOME->
AND NOT   D002000.E	// L_4th BD Z ¨¬n¡íoA¢´Ao
AND NOT   M00600	// EMERGENCY ALARM
OUT       M01512	// L_4th BD Z COMPLETE
; L12
LOAD      D001000.8	// L_4th BD Z ¢¯©ªA¢®¢¯I¡¤a
OUTP      M01513	// L_4th BD Z HOME PLS
; L13
LOAD      M01513	// L_4th BD Z HOME PLS
OR        M01514	// L_4th BD Z INITIAL HOLD
AND       D001000.8	// L_4th BD Z ¢¯©ªA¢®¢¯I¡¤a
AND NOT   M03010	// L_4th BD Z UP POS ->
AND NOT   M01515	// L_4th BD Z INITIAL ->
OUT       M01514	// L_4th BD Z INITIAL HOLD
TON       T0401 50	// L_4th BD Z GOINIT->

